# B&R Automation Studio project NAELD004C00R10L518F00 (part 33)

#### Act_Background.st
```iecst
(** 2020-05-26 **)
ACTION Act_Background:

	//Update Parameter
	IF bModuleOK = TRUE THEN

		tyParamInMove.diPosInUM		:= p_diMovePosInUM;
		tyParamInMove.diDistInUM	:= p_diMoveDistInUM;
		tyParamInMove.diVelInUMPS	:= p_diMoveVelInUMPS;
		tyParamInMove.diAcc			:= p_diMoveAcc;
		tyParamInMove.diDec			:= p_diMoveDec;

		fMotionCANUpdtDat(ADR(tyParamOut) , p_tyParamInConvert , tyParamOutDriver , tyParamInDriver , tyParamInMove , p_tyParamInHm , p_bDir, p_eNtParamMotorType);

		bWidthPosDiff	:= (tyParamOut.bIsHomed = FALSE) OR ((ABS((ABS(fAWWidthToPosInUM(p_diGoWidth , p_diWidthAtHmPos))) - tyParamOut.diActualPosInUM)) > 500);

		p_tyParamInConvert.diPitchInUM	:= fPitchCalc(p_diWidthOffsetInUM , p_diMaxWidthInUM , p_diMinWidthInUM , p_diPitchInUM);

		fbFullMovAbsBl.tyParamInConvert					:= p_tyParamInConvert;

		IF p_bDir = TRUE THEN
			bOpenSen	:= tyParamOut.bFwdLmtSen;
			bCloseSen	:= tyParamOut.bRevLmtSen;
		ELSE
			bOpenSen	:= tyParamOut.bRevLmtSen;
			bCloseSen	:= tyParamOut.bFwdLmtSen;
		END_IF

		CASE p_eNtParamMotorType OF
			DeltaAsdaA2:
				CASE tyParamOut.udiAxisErrID OF
					8976:	sAxisErrTxt	:= 'Over Current';
					12560:	sAxisErrTxt	:= 'Over Voltage';
					12576:	sAxisErrTxt	:= 'Under Voltage';
					12592:	sAxisErrTxt	:= 'Input Power Phase Loss';
					12816:	sAxisErrTxt	:= 'Regeneration Error';
					12848:	sAxisErrTxt	:= 'Overload';
					12849:	sAxisErrTxt	:= 'Pre-overload Warning';
					13056:	sAxisErrTxt	:= 'U,V,W Wiring Error';
					16912:	sAxisErrTxt	:= 'IGBT Temperature Error';
					21296:	sAxisErrTxt	:= 'Memory Error';
					21569:	sAxisErrTxt	:= 'Emergency Stop Activated';
					21570:	sAxisErrTxt	:= 'Forward Limit Switch Error';
					21571:	sAxisErrTxt	:= 'Reverse Limit Switch Error';
					21572:	sAxisErrTxt	:= 'Forward Software Limit';
					21573:	sAxisErrTxt	:= 'Reverse Software Limit';
					21760:	sAxisErrTxt	:= 'DSP Firmware Upgrade';
					25088:	sAxisErrTxt	:= 'CANopen SYNC Error';
					25360:	sAxisErrTxt	:= 'CANopen Data Initial Error';
					25376:	sAxisErrTxt	:= 'Adjustment Error';
					28961:	sAxisErrTxt	:= 'Motor Protection Error';
					28962:	sAxisErrTxt	:= 'Motor Error';
					29445:	sAxisErrTxt	:= 'Encoder Error';
					29446:	sAxisErrTxt	:= 'Encoder Output Error';
					29968:	sAxisErrTxt	:= 'Serial Communication Error';
					29984:	sAxisErrTxt	:= 'Serial Communication Time Out';
					33024:	sAxisErrTxt	:= 'CANbus Error (Bus-off)';
					33040:	sAxisErrTxt	:= 'CANopen SDO receive buffer overrun';
					33056:	sAxisErrTxt	:= 'CANbus Error (Warning)';
					33072:	sAxisErrTxt	:= 'Node Guarding or Heartbeat Error';
					33280:	sAxisErrTxt	:= 'CANopen PDO Object Error';
					33792:	sAxisErrTxt	:= 'Over Speed';
					34304:	sAxisErrTxt	:= 'Abnormal Pulse Control Command';
					34320:	sAxisErrTxt	:= 'Full Closed Loop Excessive Deviation';
					34321:	sAxisErrTxt	:= 'Excessive Deviation';
				END_CASE

			SchneiderLexium28:
				CASE tyParamOut.udiAxisErrID OF
					8724:	sAxisErrTxt	:= 'Over Current';
					8976:	sAxisErrTxt	:= 'Motor Overload';
					8977:	sAxisErrTxt	:= 'Drive overload (foldback)';
					9088:	sAxisErrTxt	:= 'Calculated offsets for current sensors out OF range';
					9089:	sAxisErrTxt := 'Motor phase missing';
					9090:	sAxisErrTxt := 'Overcurrent detected at one OF the digital outputs';
					12560:	sAxisErrTxt	:= 'DC Bus Over Voltage';
					12576:	sAxisErrTxt	:= 'DC Bus Under Voltage';
					12672:	sAxisErrTxt	:= 'Braking Resistor Overload';
					12673:	sAxisErrTxt	:= 'Safety function Safe Torque Off (STO) triggered';
					12674:	sAxisErrTxt	:= 'DC bus voltage measurement';
					12675:	sAxisErrTxt	:= 'Missing mains supply, undervoltage mains supply';
					12676:	sAxisErrTxt := 'The encoder supply voltage has dropped under operational value';
					12677:	sAxisErrTxt := 'The multi turn encoder battery voltage has dropped under 3 Vdc';
					12678:	sAxisErrTxt := 'Internal position synchronization error	detected between the multi turn AND the single turn modules';
					12679:	sAxisErrTxt := 'Generic error code of the multi turn module is detected';
					12697:	sAxisErrTxt := 'Braking resistor overload';
					16512:	sAxisErrTxt	:= 'Drive overtemperature (IPM)';
					16513:	sAxisErrTxt	:= 'Drive overtemperature (controller)';
					16534:	sAxisErrTxt := 'Temperature sensor inoperative';
					17168:	sAxisErrTxt	:= 'Power stage overtemperature';
					17280:	sAxisErrTxt := 'The encoder temperature is too high';
					17424:	sAxisErrTxt	:= 'Motor overtemperature';
					21808:	sAxisErrTxt	:= 'System error detected (nonvolatilememory)';
					21893:	sAxisErrTxt	:= 'Error detected in non-volatile memory';
					21889:	sAxisErrTxt	:= 'System error detected (nonvolatile memory)';
					21890:	sAxisErrTxt	:= 'System error detected (CAN power supply)';
					21891:	sAxisErrTxt	:= 'System error detected (selftest)';
					21894:	sAxisErrTxt	:= 'System error detected (NV ACCESS)';
					25472:	sAxisErrTxt	:= 'Target position rejected';
					25985:	sAxisErrTxt	:= 'System error detected(FPGA)';
					28816:	sAxisErrTxt	:= 'System error detected (FPGA does NOT match firmware)';
					28817:	sAxisErrTxt	:= 'Emergency Stop Activated';
					28961:	sAxisErrTxt := 'Motor blocked';
					29080:	sAxisErrTxt := 'Commutation error detected';
					29568:  sAxisErrTxt	:= 'Error detected in communication with motor encoder';
					29574:	sAxisErrTxt	:= 'Drive is not synchronous wit master cycle';
					29581:	sAxisErrTxt := 'System error detected (encoder)';
					29587:	sAxisErrTxt	:= 'Encoder overvoltage or overcurrent';
					29592:	sAxisErrTxt := 'The returned position value are no longer considered valid';
					29593:	sAxisErrTxt := 'The multi turn encoder requires an explicit configuration command';
					30081:	sAxisErrTxt := 'Target position rejected';
					30082:	sAxisErrTxt := 'No target values received via the fieldbus';
					33072:	sAxisErrTxt	:= 'CANopen: Heartbeat error detected';
					33296:	sAxisErrTxt := 'R_PDO is too short';
					33921:	sAxisErrTxt	:= 'Actual Motor Velocity Too High';
					33553:	sAxisErrTxt	:= 'Motor torque too high FOR an excessive period OF time';
					33664:	sAxisErrTxt := 'Unstable current loop';
					33922:	sAxisErrTxt := 'Velocity deviation too high';
					34321:	sAxisErrTxt	:= 'Position deviation too high';
					34432:	sAxisErrTxt := 'Position deviation via signal output function MC_OK';
					34441:	sAxisErrTxt := 'Position deviation too high (following error)';
					61568:	sAxisErrTxt	:= 'Fieldbus: Communication	error detected';
					65282:	sAxisErrTxt	:= 'Not possible to read data of electronic motor nameplate';
					65296:	sAxisErrTxt	:= 'Forward Limit Switch Error';
					65297:	sAxisErrTxt	:= 'Reverse Limit Switch Error';
					65281:	sAxisErrTxt := 'System error detected';
					65298:	sAxisErrTxt	:= 'Forward Software Limit';
					65299:	sAxisErrTxt	:= 'Reverse Software Limit';
					65301:	sAxisErrTxt := 'The encoder firmware cannot operate on the provided hardware';

				END_CASE

			EstunPronet:
				CASE tyParamOut.udiAxisErrID OF
					65281:	sAxisErrTxt	:= 'Parameter breakdown';//A01
					65282:	sAxisErrTxt	:= 'AD shift channels breakdown';
					65283:	sAxisErrTxt	:= 'Overspeed';
					65284:	sAxisErrTxt	:= 'Overload';
					65285:	sAxisErrTxt := 'Position error counteroverflow ';
					65286:	sAxisErrTxt := 'Position error pulse overflow';
					65287:	sAxisErrTxt	:= 'The setting of electronic gear or given pulse frequency is not reasonable';
					65288:	sAxisErrTxt	:= 'The 1st channel of current detection is wrong.';
					65289:	sAxisErrTxt	:= 'The 2nd channel of current detection is wrong.';
					65290:	sAxisErrTxt	:= 'Incremental Encoder is break off.';//A10
					65292:	sAxisErrTxt	:= 'Overcurrent';
					65293:	sAxisErrTxt	:= 'Overvoltage';
					65294:	sAxisErrTxt	:= 'Undervoltage';
					65295:	sAxisErrTxt := 'Bleeder resistor error';
					65296:	sAxisErrTxt := 'Regeneration error';
					65297:	sAxisErrTxt := 'Resolver error';
					65298:	sAxisErrTxt := 'IGBT superheat alarm';
					65299:	sAxisErrTxt := 'Motor overheat alarm';
					65300:	sAxisErrTxt := 'Power line phase shortage';//A20
					65301:	sAxisErrTxt	:= 'Instantaneous power off alarm';
					65302:	sAxisErrTxt	:= 'Motor temperature detection sensor is break off.';
					65303:	sAxisErrTxt := 'Brake overcurrent alarm';//A23
					65305:	sAxisErrTxt := 'Motor power line U overcurrent';//A25
					65306:	sAxisErrTxt := 'Motor power line V overcurrent';//A26
					65307:	sAxisErrTxt := 'Motor power line W overcurrent';//A27
					65322:	sAxisErrTxt	:= 'Servomotor type error';//A42
					65323:	sAxisErrTxt	:= 'Servo drive type error';
					65325:	sAxisErrTxt	:= 'Absolute encoder multiturn information error';
					65326:	sAxisErrTxt	:= 'Absolute encoder multiturn information overflow';
					65327:	sAxisErrTxt	:= 'Battery voltage below 2.5V';
					65328:	sAxisErrTxt	:= 'Battery voltage below 3.1V';//A48
					65330:	sAxisErrTxt := 'Serial encoder communication overtime ';//A50
					65331:	sAxisErrTxt := 'Absolute encoder overspeed alarm detected';
					65332:  sAxisErrTxt	:= 'Absolute state of serial encoder error';
					65333:	sAxisErrTxt	:= 'Serial encoder calcaution error';
					65334:	sAxisErrTxt := 'Parity bit or end bit in serial encoder control domain error';
					65335:	sAxisErrTxt	:= 'Serial encoder communication data checking error';
					65336:	sAxisErrTxt := 'End bit in serial encoder control domain error';
					65338:	sAxisErrTxt := 'Serial encoder data empty';
					65339:	sAxisErrTxt := 'Serial encoder data format error';
					65340:	sAxisErrTxt := 'Communication module not detected ';//A60
					65341:	sAxisErrTxt := 'Communication unsuccessful';
					65342:	sAxisErrTxt := 'Servo drive can not receive the period data of communication module ';
					65343:	sAxisErrTxt := 'Communication module can not receive the servo drive response data.';
					65344:	sAxisErrTxt := 'Communication module and bus connectionless';
					65346:	sAxisErrTxt := 'CAN communication abnormal';
					65347:	sAxisErrTxt := 'Receiving heartbeat timeout';
					65349:	sAxisErrTxt := 'Synchronization signal monitoring cycle is longer than setting';
					65362: sAxisErrTxt	:= 'Torque output alarm';
				END_CASE
		END_CASE

	ELSE

		tyParamOut.bAxisErr			:= FALSE;
		tyParamOut.bFwdLmtSen		:= FALSE;
		tyParamOut.bInPos			:= FALSE;
		tyParamOut.bIsHomed			:= FALSE;
		tyParamOut.bPosDiff			:= TRUE;
		tyParamOut.bPwrOn			:= FALSE;
		tyParamOut.bRevLmtSen		:= FALSE;
		tyParamOut.bStopped			:= TRUE;
		tyParamOut.diActualPosInUM	:= 0;
		tyParamOut.diHmAcc			:= 0;
		tyParamOut.diHmSpdForSwitch	:= 0;
		tyParamOut.diHmSpdForZero	:= 0;
		tyParamOut.diProfileAcc		:= 0;
		tyParamOut.diProfileDec		:= 0;
		tyParamOut.udiAxisErrID		:= 0;

		bWidthPosDiff				:= TRUE;

	END_IF

	//Abnormal Movement
	IF eStatus1 <> Error THEN
		IF p_bOps = TRUE AND eStatus = Idle THEN
			IF (ABS(tyParamOut.diActualPosInUM - diActualPosInUMOld) > 2000) AND (ABS(tyParamOut.diActualPosInUM - diActualPosInUMOld) < 10000) THEN
				eStatus1	:= Error;
				udiStatus1	:= 10000;	//Axis Move Abnormally By External Force

				fMotionCANRstCtrlWord(ADR(tyParamOutDriver));
				p_eAct	:= AWActIdle;
				eStat	:= AWActIdle;
			END_IF
		ELSE
			diActualPosInUMOld	:= tyParamOut.diActualPosInUM;
		END_IF
	END_IF

	//Reset Error
	IF (eStatus1 = Error) AND bRstErr THEN
		eStatus1	:= Idle;
		udiStatus1	:= 0;
	END_IF

	//Request Position To Movement Out Of Range
	IF p_bOps
		AND((tyParamInMove.diPosInUM < p_diMinAbsPosInUM) OR (tyParamInMove.diPosInUM > p_diMaxAbsPosInUM))
		AND (eStatus2 <> Error) THEN
		eStatus2	:= Error;
		udiStatus2	:= 10029;	//Request Absolute Position Out Of Range

		fMotionCANRstCtrlWord(ADR(tyParamOutDriver));
		p_eAct	:= AWActIdle;
		eStat	:= AWActIdle;
	END_IF

	//Reset Error
	IF (eStatus2 = Error) AND bRstErr THEN
		eStatus2	:= Idle;
		udiStatus2	:= 0;
	END_IF

	//Sensor Interrupt
	IF (bNotInterruptible = TRUE OR bJogging) AND eStatus3 <> Error THEN

		IF p_bInletSensor = TRUE THEN
			eStatus3	:= Error;
			udiStatus3	:= 10030;	//Inlet Sensor Interrupt Auto Width Movement

			fMotionCANRstCtrlWord(ADR(tyParamOutDriver));
			p_eAct	:= AWActIdle;
			eStat	:= AWActIdle;

		ELSIF p_bOutletSensor = TRUE THEN
			eStatus3	:= Error;
			udiStatus3	:= 10031;	//Outlet Sensor Interrupt Auto Width Movement

			fMotionCANRstCtrlWord(ADR(tyParamOutDriver));
			p_eAct	:= AWActIdle;
			eStat	:= AWActIdle;

		ELSIF p_bClearSensor = TRUE THEN
			eStatus3	:= Error;
			udiStatus3	:= 10032;	//Clear Sensor Interrupt Auto Width Movement

			fMotionCANRstCtrlWord(ADR(tyParamOutDriver));
			p_eAct	:= AWActIdle;
			eStat	:= AWActIdle;

		ELSIF p_bMiddleSensor = TRUE THEN
			eStatus3	:= Error;
			udiStatus3	:= 10033;	//Middle Sensor Interrupt Auto Width Movement

			fMotionCANRstCtrlWord(ADR(tyParamOutDriver));
			p_eAct	:= AWActIdle;
			eStat	:= AWActIdle;

		ELSIF p_bInterruptSensor = TRUE THEN
			eStatus3	:= Error;
			udiStatus3	:= 10034;	//Sensor Interrupt Auto Width Movement

			fMotionCANRstCtrlWord(ADR(tyParamOutDriver));
			p_eAct	:= AWActIdle;
			eStat	:= AWActIdle;

		ELSIF p_bCloseInterruptSensor = TRUE AND bJogOpen = FALSE THEN
			eStatus3	:= Error;
			udiStatus3	:= 10047;	//Sensor Interrupt Auto Width Movement

			fMotionCANRstCtrlWord(ADR(tyParamOutDriver));
			p_eAct	:= AWActIdle;
			eStat	:= AWActIdle;

		ELSIF p_bOpenInterruptSensor = TRUE AND bJogClose = FALSE THEN
			eStatus3	:= Error;
			udiStatus3	:= 10048;	//Sensor Interrupt Auto Width Movement

			fMotionCANRstCtrlWord(ADR(tyParamOutDriver));
			p_eAct	:= AWActIdle;
			eStat	:= AWActIdle;
		END_IF

	END_IF

	//Reset Error
	IF (eStatus3 = Error AND bRstErr)
		OR (p_bOpenInterruptSensor AND eStat = AWActJogClose)
		OR (p_bCloseInterruptSensor AND eStat = AWActJogOpen)
		THEN
		eStatus3	:= Idle;
		udiStatus3	:= 0;
	END_IF

	IF bRstErr THEN
		udiStatus	:= 0;
		bJogging	:= FALSE;
		bJogClose	:= FALSE;
		bJogOpen	:= FALSE;
	END_IF

	fbServoModuleOk(IN:= bModuleOK);
	fbServoModuleNotOk(IN:= bModuleOK = FALSE);
	IF fbServoModuleNotOk.Q AND udiStatus <> 10001 THEN

		bModuleNotOK		:= TRUE;
		bModuleNotOKLock	:= TRUE;
		usiRstStep	:= 0;
		tyParamOutDriver.uiCtrlword_6040	:= 0;
		tyParamOutDriver.siModOfOpt_6060	:= 0;
		tyParamOutDriver.diTargetPos_607A	:= 0;
		tyParamOutDriver.udiMoveSpd_6081	:= 0;
		tyParamOutDriver.siHmMethod_6098	:= 0;
		tyParamOutDriver.diJogVel_60FF		:= 0;

		CASE p_eNtParamMotorType OF

			DeltaAsdaA2:
				fbModuleOK(bModuleOK:= FALSE);
				IF eStatus = Idle THEN
					eAct	:= AWActRstNode;
				END_IF

				IF (eStatus = Done OR eStatus = Error)AND eStat = AWActRstNode THEN

					eAct	:= AWActIdle;
				END_IF

			EstunPronet:
				fbModuleOK(bModuleOK:= FALSE);
				IF eStatus = Idle THEN
					eAct	:= AWActRstNode;
				END_IF

				IF (eStatus = Done OR eStatus = Error)AND eStat = AWActRstNode THEN

					eAct	:= AWActIdle;
				END_IF

			SchneiderLexium28:
			// Do Nothing
		END_CASE

	ELSIF bModuleNotOK = TRUE AND fbServoModuleOk.Q THEN

		CASE usiRstStep OF

			0:
				IF eStatus = Idle THEN
					eAct	:= AWActRstAxisErr;
				END_IF

				IF eStatus = Done AND eStat = AWActRstAxisErr THEN
					eAct	:= AWActIdle;
					usiRstStep	:= 4;
				END_IF

			4: tyParamOutDriver.siModOfOpt_6060 := 1;
				usiRstStep	:= 5;

			5: tyParamOutDriver.siModOfOpt_6060 := 1;
				fbRstNodeTimer(IN:=TRUE);

				IF tyParamInDriver.siModOfOptDisp_6061 = 1 THEN
					usiRstStep	:= 6;
					fbRstNodeTimer(IN:=FALSE);
				ELSIF fbRstNodeTimer.Q THEN
					usiRstStep	:= 8;
					fbRstNodeTimer(IN:=FALSE);
				END_IF

			6: tyParamOutDriver.siModOfOpt_6060 := 6;
				fbRstNodeTimer(IN:=FALSE);
				usiRstStep	:= 7;

			7: tyParamOutDriver.siModOfOpt_6060 := 6;
				fbRstNodeTimer(IN:=TRUE);

				IF tyParamInDriver.siModOfOptDisp_6061 = 6 THEN
					usiRstStep	:= 10;
					fbRstNodeTimer(IN:=FALSE);
				ELSIF fbRstNodeTimer.Q THEN
					usiRstStep	:= 9;
					fbRstNodeTimer(IN:=FALSE);
				END_IF

			8:	fbModuleOK(bEn := TRUE, bModuleOK:= FALSE);
				fbRstNodeTimer(IN:=FALSE);
				usiRstStep	:= 9;

			9:	fbModuleOK(bModuleOK:= FALSE);
				IF eStatus = Idle THEN
					eAct	:=AWActRstNode;
				END_IF

				IF eStatus = Done AND eStat = AWActRstNode THEN
					usiRstStep	:= 0;
					eAct		:= AWActIdle;
				END_IF

			10:IF eStatus = Idle THEN
					eAct	:= AWActRstAxisErr;
				END_IF

				IF eStatus = Done AND eStat = AWActRstAxisErr THEN
					eAct			:=AWActIdle;
					usiRstStep	:= 11;
				END_IF

			11:

				IF eStatus = Idle THEN
					eAct	:= AWActSDOWrite;
				END_IF

				IF eStatus = Done AND eStat = AWActSDOWrite THEN
					eAct			:= AWActIdle;
					usiRstStep	:= 13;

				ELSIF udiStatus = 10028 THEN
					eAct			:= AWActIdle;
					usiRstStep	:= 0;
				END_IF

			13: bModuleNotOK	:= FALSE;
				usiRstStep	:= 0;
		END_CASE
	ELSE
		eAct	:= AWActIdle;

	END_IF

	IF tyParamOut.bPosDiff = FALSE THEN
		tyParamOutDriver.uiCtrlword_6040.4	:= FALSE;
	END_IF

END_ACTION
```

#### Act_InitGlobal.st
```iecst
(** 2019-04-09 **)
ACTION Act_InitGlobal:

	(* Always Change If Project Change *)

	//Pass Data To Link
	p_bLinkOpsRun ACCESS p_OpsRun;
	p_bLinkStartupRun ACCESS p_StartupRun;
	p_diLinkProdSelWidth ACCESS p_ProdRcpCurrRcp2Width;
	p_diLinkPshrOffset ACCESS p_ProdRcpCurrRcp2PshrOffset;
	p_diLinkMnlGoWidth ACCESS p_UIMnlAWPushOrPullerGoWidth;
	p_bLinkSafetyRelay ACCESS p_DISafetyRlySig;

	//Pass Data To Internal Use
	p_udiRstErr ACCESS p_RstErrReset;
	p_bManual ACCESS p_UIMnlMod;
	p_bEn ACCESS p_DISimServoEn;
	p_bPrep ACCESS p_NtParamAWPusherPrep;
	p_bDis ACCESS p_McParamAWPusherDis;
	p_bOps ACCESS p_OpsStatusRun;
	p_diWidthAtHmPos ACCESS p_McParamAWPusherAtHmPos;
	p_tyTuning ACCESS p_NtParamAWPushPulTuning;
	p_diJogVelInUMPS ACCESS p_UIMnlAWPushOrPullerJogSpd;
	p_diMovePosInUM ACCESS p_UIMnlAWPushOrPullerTargetPos;
	p_diMoveDistInUM ACCESS p_UIMnlAWPushOrPullerStepSize;
	p_bUITeachServo ACCESS p_UITeachServo;
	p_diMoveAcc ACCESS p_NtParamAWPushPulAcc;
	p_diMoveDec ACCESS p_NtParamAWPushPulDec;
	p_diMinWidthInUM ACCESS p_NtParamProdRcpMinWidth;
	p_diMaxWidthInUM ACCESS p_NtParamProdRcpMaxWidth;
	p_diWidthOffsetInUM ACCESS p_NtParamPushPulAWidthOffset;
	p_bInletSensor ACCESS p_DIConvLftSen;
	p_bOutletSensor ACCESS p_DIConvRgtSen;
	p_bDir ACCESS p_NtParamAWPushPulDir;
	p_bDirBl ACCESS p_NtParamAWPushPulDirBl;
	p_usiNode ACCESS p_NtParamAWPushPulNode;
	p_sDevice ACCESS p_NtParamAWPushPulDevice;
	p_sProgNm ACCESS p_NtParamAWPushPulProgNm;
	p_diMoveBacklashDistInUM ACCESS p_NtParamAWPushPulMovBlDistInUM;
	p_diPitchInUM ACCESS p_NtParamAWPushPulPitchInUM;
	p_tyParamInHm ACCESS p_NtParamAWPushPulParamInHm;
	p_tyParamInConvert ACCESS p_NtParamAWPushPulParamInConvert;
	p_bNtSettingsLoadDone ACCESS p_StartupNtSettingsLoadDone;
	p_eNtParamMotorType ACCESS p_NtParamAWPushPulMotorType;

	p_bInletShutterCloseRS ACCESS p_DIInShutterCloseRS;
	p_bOutletShutterCloseRS ACCESS p_DIOutShutterCloseRS;
	p_bProjInletShutPrep ACCESS p_NtParamProjInletShutPrep;
	p_bProjOutletShutPrep ACCESS p_NtParamProjOutletShutPrep;
	p_bOutShutterDis ACCESS p_McParamOutShutterDis;
	p_bPullerRetSen ACCESS p_DIPullerRetRS;
	p_bPullerExtSen ACCESS p_DIPullerExtRS;
	(* Always Change If Project Change *)

END_ACTION
```

#### Act_Link.st
```iecst
(** 2019-03-29 **)
ACTION Act_Link:

	IF p_bManual = TRUE THEN
		p_diMoveVelInUMPS ACCESS p_UIMnlAWPushOrPullerNomSpd;
		IF p_diLinkMnlGoWidth < p_diWidthAtHmPos THEN
			p_diGoWidth := p_diWidthAtHmPos;
		ELSE
			p_diGoWidth	:= p_diLinkMnlGoWidth;
		END_IF

	ELSE

		p_diMoveVelInUMPS ACCESS p_NtParamAWPushPulAutoSpd;
		IF ((p_diLinkProdSelWidth/2) + p_diLinkPshrOffset) < p_diWidthAtHmPos THEN
			p_diGoWidth := p_diWidthAtHmPos+3000;
		ELSE
			//	p_diGoWidth := ((p_diLinkProdSelWidth/2) + p_diLinkPshrOffset)/2;
			IF p_diLinkPshrOffset = 0 THEN
				p_diGoWidth := (p_diLinkProdSelWidth/2) - 50000;
			ELSE
				p_diGoWidth := (p_diLinkProdSelWidth/2) + p_diLinkPshrOffset;
			END_IF
		END_IF

	END_IF

	IF p_bProjInletShutPrep = TRUE THEN
		IF p_bInletShutterCloseRS = FALSE OR p_bPullerRetSen = FALSE
			THEN
			bInterruptSensor1 := TRUE;
		ELSE
			bInterruptSensor1 := FALSE;
		END_IF
	ELSE
		bInterruptSensor1 := FALSE;
	END_IF

	IF p_bProjOutletShutPrep = TRUE AND p_bOutShutterDis = FALSE THEN
		IF p_bOutletShutterCloseRS = FALSE OR p_bPullerRetSen = FALSE
			THEN
			bInterruptSensor2 := TRUE;
		ELSE
			bInterruptSensor2 := FALSE;
		END_IF
	ELSE
		bInterruptSensor2 := FALSE;
	END_IF

	p_bInterruptSensor := bInterruptSensor2 OR bInterruptSensor1;// OR p_bLinkSafetyRelay = FALSE;

END_ACTION
```

#### Act_LinkAction.st
```iecst
(** 2019-10-21 **)
ACTION Act_LinkAction:

	IF eStatus = Idle THEN
		IF bModuleNotOK THEN
			p_eAct ACCESS ADR(eAct);
		ELSE
			IF p_bLinkStartupRun = TRUE THEN
				p_eAct ACCESS p_StartupAWPushPulAct;
			ELSIF p_bLinkOpsRun = TRUE THEN
				p_eAct ACCESS p_OpsTravLifLDAWPushPullAct;
			ELSIF p_bManual = TRUE THEN
				p_eAct ACCESS p_UIAWPushOrPullerAct;
			ELSE
				p_eAct ACCESS ADR(eAct);
			END_IF
		END_IF
	END_IF

	IF EDGENEG(p_bManual) OR EDGENEG(p_bLinkOpsRun) OR EDGENEG(p_bLinkStartupRun) THEN
		tyParamOutDriver.uiCtrlword_6040	:= 0;
	END_IF

END_ACTION
```

### Program Logical/CANOpenServo/Trav/Trav

#### InputRef.var
```iecst
(*2020-03-16*)
(**)
(*General*)
VAR
	p_eAct : REFERENCE TO eTravAction;
	p_udiRstErr : REFERENCE TO UDINT;
	p_bPrep : REFERENCE TO BOOL;
	p_bEn : REFERENCE TO BOOL;
	p_bDis : REFERENCE TO BOOL;
END_VAR
(**)
(*Configuration*)
VAR
	p_bOps : REFERENCE TO BOOL;
	p_bManual : REFERENCE TO BOOL;
	p_diAPos : REFERENCE TO DINT;
	p_diBPos : REFERENCE TO DINT;
	p_diCPos : REFERENCE TO DINT;
	p_diDPos : REFERENCE TO DINT;
	p_diEPos : REFERENCE TO DINT;
	p_diFPos : REFERENCE TO DINT;
	p_diGPos : REFERENCE TO DINT;
	p_diHPos : REFERENCE TO DINT;
	p_tyTuning : REFERENCE TO tyMotionCANTuning;
	p_diJogVelInUMPS : REFERENCE TO DINT;
	p_diMovePosInUM : REFERENCE TO DINT;
	p_diMoveDistInUM : REFERENCE TO DINT;
	p_diMoveVelInUMPS : REFERENCE TO DINT;
	p_diMoveAcc : REFERENCE TO DINT;
	p_diMoveDec : REFERENCE TO DINT;
	p_diMinAbsPosInUM : REFERENCE TO DINT;
	p_diMaxAbsPosInUM : REFERENCE TO DINT;
	p_bInterruptSensor1 : REFERENCE TO BOOL;
	p_bInterruptSensor2 : REFERENCE TO BOOL;
	p_bInterruptSensor3 : REFERENCE TO BOOL;
	p_bInterruptSensor4 : REFERENCE TO BOOL;
	p_bInterruptSensor5 : REFERENCE TO BOOL;
	p_usiNode : REFERENCE TO USINT;
	p_bDir : REFERENCE TO BOOL;
	p_bNoIndexPulse : REFERENCE TO BOOL;
	p_sDevice : REFERENCE TO STRING[3];
	p_sProgNm : REFERENCE TO STRING[15];
	p_tyParamInHm : REFERENCE TO tyMotionCANParamInHm;
	p_tyParamInConvert : REFERENCE TO tyMotionCANParamInConvert;
	p_bNtSettingsLoadDone : REFERENCE TO BOOL;
	p_eNtParamMotorType : REFERENCE TO eServoMotorType;
	p_bProjInletShutPrep : REFERENCE TO BOOL;
	p_bProjOutletShutPrep : REFERENCE TO BOOL;
	p_bOutletShutterCloseRS : REFERENCE TO BOOL;
	p_bOutShutterDis : REFERENCE TO BOOL;
	p_bInletShutterCloseRS : REFERENCE TO BOOL;
	p_bPullerExtSen : REFERENCE TO BOOL;
	p_bPullerRetSen : REFERENCE TO BOOL;
	p_bPullerRotHmRS : REFERENCE TO BOOL;
	p_bDIConvClrSen : REFERENCE TO BOOL;
	p_bDIConvLftSen : REFERENCE TO BOOL;
END_VAR
```

#### InputRef_Link.var
```iecst
(*2019-04-09*)
(**)
(*External Data*)
VAR
	p_bLinkOpsRun : REFERENCE TO BOOL;
	p_bLinkStartupRun : REFERENCE TO BOOL;
	p_bSimu : REFERENCE TO BOOL;
	p_diLinkAPos : REFERENCE TO DINT;
	p_diLinkBPos : REFERENCE TO DINT;
	p_diLinkCPos : REFERENCE TO DINT;
	p_diLinkGPos : REFERENCE TO DINT;
	p_diLinkAPos1 : REFERENCE TO DINT;
	p_diLinkBPos1 : REFERENCE TO DINT;
	p_diLinkCPos1 : REFERENCE TO DINT;
	p_diLinkGPos1 : REFERENCE TO DINT;
	p_bLinkNtParamProjRotCylPrep : REFERENCE TO BOOL;
END_VAR
(**)
VAR
	p_eLinkMag : REFERENCE TO eLDMag;
	p_usiLinkMod : REFERENCE TO USINT;
	p_bLinkOpsTravLifULInDSPos : REFERENCE TO BOOL;
	p_bLinkOpsTravLifUSMagWidthChk : REFERENCE TO BOOL;
	p_bLinkNtParamProjDsFixToFixRail : REFERENCE TO BOOL;
	p_diLinkFixtoFixPosIn : REFERENCE TO DINT;
	p_diLinkMcParamTravPosB : REFERENCE TO DINT;
	p_tyProdRcpCurrRcp : REFERENCE TO tyProdRcpParam;
	p_bLinkSafetyRelay : REFERENCE TO BOOL;
	p_bLinkProjLifterMagPlatform : REFERENCE TO BOOL;
	p_bLinkTravGotoChkPt : REFERENCE TO BOOL;
	p_diLinkTravGotoChkPtDist1 : REFERENCE TO DINT;
	p_diLinkTravGotoChkPtDist2 : REFERENCE TO DINT;
	p_diLinkTravGotoChkPtDist3 : REFERENCE TO DINT;
	p_diLaneBOffset : REFERENCE TO DINT;
END_VAR
```

#### Local.var
```iecst
(*2020-03-16*)
(**)
(*Local Action, State & Status*)
VAR
	eAct : eTravAction := TravActIdle;
	eStat : eTravAction := TravActIdle;
	eMainStatus : eFBStatus := Idle;
	eStatus : eFBStatus := Idle;
	eStatus1 : eFBStatus := Idle;
	eStatus2 : eFBStatus := Idle;
	eStatus3 : eFBStatus := Idle;
	udiStatus : UDINT := 0;
	udiStatus1 : UDINT := 0;
	udiStatus2 : UDINT := 0;
	udiStatus3 : UDINT := 0;
	sStatTxt : STRING[200] := '';
	a_sStatText : ARRAY[0..50] OF STRING[200] := ['Idling','Going A Position','Going B Position','Going C Position','Going D Position','Going E Position','Going F Position','Going G Position','Going H Position','Full Homing','Powering On','Powering Off','Homing','Moving Absolute','Moving Relative','Jogging Front','Jogging Rear','Jogging Stop','Resetting Axis Error','Stopping','Writing SDO','Background Start Module OK Check','Background Stop Module OK Check',28('')];
END_VAR
(**)
(*Local Alarm*)
VAR
	tyAlmData : tyAlmDat;
	tyAlmData1 : tyAlmDat;
	tyAlmData2 : tyAlmDat;
	tyAlmData3 : tyAlmDat;
	a_tyAlmText : ARRAY[10000..10299] OF tyAlmTxt := [(sAlmText:='Axis Move Abnormally By External Force',sRcyText:='Servo Motor Abnormal Operation. Reset And Resume Operation. If The Problem Persists, Please Contact Nutek For A Possible Solution.'),(sAlmText:='CANOpen Communication Error, ModuleOK Not TRUE',sRcyText:='Fail While Read/Write Data. Reset The Error And Resume Operation.'),(sAlmText:='Power On Time Out While Going A Position',sRcyText:='Timeout Expired Before Operation Completed. Reset And Resume Operation.'),(sAlmText:='Homing Time Out While Going A Position',sRcyText:='Timeout Expired Before Operation Completed. Reset And Resume Operation.'),(sAlmText:='Move Absolute Time Out While Going A Position',sRcyText:='Timeout Expired Before Operation Completed. Reset And Resume Operation.'),(sAlmText:='Stop Motion Time Out While Going A Position',sRcyText:='Timeout Expired Before Operation Completed. Reset And Resume Operation.'),(sAlmText:='Axis Error Reset Failed While Going A Position',sRcyText:='Axis Error Reset Failed. Please Retry Again Reset Operation. If The Problem Persists, Please Contact Nutek For A Possible Solution.'),(sAlmText:='Axis Error Occur In Move Absolute While Going A Position',sRcyText:='Servo Motor Abnormal Operation. Reset And Resume Operation. If The Problem Persists, Please Contact Nutek For A Possible Solution.'),(sAlmText:='Axis Error Occur In Homing While Going A Position',sRcyText:='Servo Motor Abnormal Operation. Reset And Resume Operation. If The Problem Persists, Please Contact Nutek For A Possible Solution.'),(sAlmText:='Homing Done But Home Flag Is Not Activated While Going A Position',sRcyText:='Servo Motor Abnormal Operation. Reset And Resume Operation. If The Problem Persists, Please Contact Nutek For A Possible Solution.'),(sAlmText:='Forward Limit Activated In Homing While Going A Position',sRcyText:='Forward Limit Switch Is Activated. Reset The Error By Operate The Motor Backwards.'),(sAlmText:='Reverse Limit Activated In Homing While Going A Position',sRcyText:='Reverse Limit Switch Is Activated. Reset The Error By Operate The Motor Backwards.'),(sAlmText:='Forward Limit Activated In Move Absolute While Going A Position',sRcyText:='Forward Limit Switch Is Activated. Reset The Error By Operate The Motor Backwards.'),(sAlmText:='Reverse Limit Activated In Move Absolute While Going A Position',sRcyText:='Reverse Limit Switch Is Activated. Reset The Error By Operate The Motor Backwards.'),(sAlmText:='Power On Time Out While Full Homing',sRcyText:='Timeout Expired Before Operation Completed. Reset And Resume Operation.'),(sAlmText:='Homing Time Out While Full Homing',sRcyText:='Timeout Expired Before Operation Completed. Reset And Resume Operation.'),(sAlmText:='Stop Motion Time Out While Full Homing',sRcyText:='Timeout Expired Before Operation Completed. Reset And Resume Operation.'),(sAlmText:='Axis Error Reset Failed While Full Homing',sRcyText:='Axis Error Reset Failed. Please Retry Again Reset Operation. If The Problem Persists, Please Contact Nutek For A Possible Solution.'),(sAlmText:='Axis Error Occur In Homing While Full Homing',sRcyText:='Servo Motor Abnormal Operation. Reset And Resume Operation. If The Problem Persists, Please Contact Nutek For A Possible Solution.'),(sAlmText:='Homing Done But Home Flag Is Not Activated While Full Homing',sRcyText:='Servo Motor Abnormal Operation. Reset And Resume Operation. If The Problem Persists, Please Contact Nutek For A Possible Solution.'),(sAlmText:='Forward Limit Activated In Homing While Full Homing',sRcyText:='Forward Limit Switch Is Activated. Reset The Error By Operate The Motor Backwards.'),(sAlmText:='Reverse Limit Activated In Homing While Full Homing',sRcyText:='Reverse Limit Switch Is Activated. Reset The Error By Operate The Motor Backwards.'),(sAlmText:='Power On Time Out',sRcyText:='Timeout Expired Before Operation Completed. Reset And Resume Operation.'),(sAlmText:='Power Off Time Out',sRcyText:='Timeout Expired Before Operation Completed. Reset And Resume Operation.'),(sAlmText:='Homing Time Out',sRcyText:='Timeout Expired Before Operation Completed. Reset And Resume Operation.'),(sAlmText:='Move Absolute Time Out',sRcyText:='Timeout Expired Before Operation Completed. Reset And Resume Operation.'),(sAlmText:='Move Relative Time Out',sRcyText:='Timeout Expired Before Operation Completed. Reset And Resume Operation.'),(sAlmText:='Stop Motion Time Out',sRcyText:='Timeout Expired Before Operation Completed. Reset And Resume Operation.'),(sAlmText:='SDO Write Error',sRcyText:='Fail While Write Data. Reset The Error And Resume Operation.'),(sAlmText:='Power On Time Out While Going B Position',sRcyText:='Timeout Expired Before Operation Completed. Reset And Resume Operation.'),(sAlmText:='Homing Time Out While Going B Position',sRcyText:='Timeout Expired Before Operation Completed. Reset And Resume Operation.'),(sAlmText:='Move Absolute Time Out While Going B Position',sRcyText:='Timeout Expired Before Operation Completed. Reset And Resume Operation.'),(sAlmText:='Stop Motion Time Out While Going B Position',sRcyText:='Timeout Expired Before Operation Completed. Reset And Resume Operation.'),(sAlmText:='Axis Error Reset Failed While Going B Position',sRcyText:='Axis Error Reset Failed. Please Retry Again Reset Operation. If The Problem Persists, Please Contact Nutek For A Possible Solution.'),(sAlmText:='Axis Error Occur In Move Absolute While Going B Position',sRcyText:='Servo Motor Abnormal Operation. Reset And Resume Operation. If The Problem Persists, Please Contact Nutek For A Possible Solution.'),(sAlmText:='Axis Error Occur In Homing While Going B Position',sRcyText:='Servo Motor Abnormal Operation. Reset And Resume Operation. If The Problem Persists, Please Contact Nutek For A Possible Solution.'),(sAlmText:='Homing Done But Home Flag Is Not Activated While Going B Position',sRcyText:='Servo Motor Abnormal Operation. Reset And Resume Operation. If The Problem Persists, Please Contact Nutek For A Possible Solution.'),(sAlmText:='Forward Limit Activated In Homing While Going B Position',sRcyText:='Forward Limit Switch Is Activated. Reset The Error By Operate The Motor Backwards.'),(sAlmText:='Reverse Limit Activated In Homing While Going B Position',sRcyText:='Reverse Limit Switch Is Activated. Reset The Error By Operate The Motor Backwards.'),(sAlmText:='Forward Limit Activated In Move Absolute While Going B Position',sRcyText:='Forward Limit Switch Is Activated. Reset The Error By Operate The Motor Backwards.'),(sAlmText:='Reverse Limit Activated In Move Absolute While Going B Position',sRcyText:='Reverse Limit Switch Is Activated. Reset The Error By Operate The Motor Backwards.'),(sAlmText:='Sensor Interrupt Movement',sRcyText:='Clear Interrupt Sensor And Resume Operation.'),35((0)),(sAlmText:='Request Absolute Position Out Of Range',sRcyText:='Request Absolute Position Does Not Fall Within The Expected Range.'),(sAlmText:='Power On Time Out While Going C Position',sRcyText:='Timeout Expired Before Operation Completed. Reset And Resume Operation.'),(sAlmText:='Homing Time Out While Going C Position',sRcyText:='Timeout Expired Before Operation Completed. Reset And Resume Operation.'),(sAlmText:='Move Absolute Time Out While Going C Position',sRcyText:='Timeout Expired Before Operation Completed. Reset And Resume Operation.'),(sAlmText:='Stop Motion Time Out While Going C Position',sRcyText:='Timeout Expired Before Operation Completed. Reset And Resume Operation.'),(sAlmText:='Axis Error Reset Failed While Going C Position',sRcyText:='Axis Error Reset Failed. Please Retry Again Reset Operation. If The Problem Persists, Please Contact Nutek For A Possible Solution.'),(sAlmText:='Axis Error Occur In Move Absolute While Going C Position',sRcyText:='Servo Motor Abnormal Operation. Reset And Resume Operation. If The Problem Persists, Please Contact Nutek For A Possible Solution.'),(sAlmText:='Axis Error Occur In Homing While Going C Position',sRcyText:='Servo Motor Abnormal Operation. Reset And Resume Operation. If The Problem Persists, Please Contact Nutek For A Possible Solution.'),(sAlmText:='Homing Done But Home Flag Is Not Activated While Going C Position',sRcyText:='Servo Motor Abnormal Operation. Reset And Resume Operation. If The Problem Persists, Please Contact Nutek For A Possible Solution.'),(sAlmText:='Forward Limit Activated In Homing While Going C Position',sRcyText:='Forward Limit Switch Is Activated. Reset The Error By Operate The Motor Backwards.'),(sAlmText:='Reverse Limit Activated In Homing While Going C Position',sRcyText:='Reverse Limit Switch Is Activated. Reset The Error By Operate The Motor Backwards.'),(sAlmText:='Forward Limit Activated In Move Absolute While Going C Position',sRcyText:='Forward Limit Switch Is Activated. Reset The Error By Operate The Motor Backwards.'),(sAlmText:='Reverse Limit Activated In Move Absolute While Going C Position',sRcyText:='Reverse Limit Switch Is Activated. Reset The Error By Operate The Motor Backwards.'),(sAlmText:='Power On Time Out While Going D Position',sRcyText:='Timeout Expired Before Operation Completed. Reset And Resume Operation.'),(sAlmText:='Homing Time Out While Going D Position',sRcyText:='Timeout Expired Before Operation Completed. Reset And Resume Operation.'),(sAlmText:='Move Absolute Time Out While Going D Position',sRcyText:='Timeout Expired Before Operation Completed. Reset And Resume Operation.'),(sAlmText:='Stop Motion Time Out While Going D Position',sRcyText:='Timeout Expired Before Operation Completed. Reset And Resume Operation.'),(sAlmText:='Axis Error Reset Failed While Going D Position',sRcyText:='Axis Error Reset Failed. Please Retry Again Reset Operation. If The Problem Persists, Please Contact Nutek For A Possible Solution.'),(sAlmText:='Axis Error Occur In Move Absolute While Going D Position',sRcyText:='Servo Motor Abnormal Operation. Reset And Resume Operation. If The Problem Persists, Please Contact Nutek For A Possible Solution.'),(sAlmText:='Axis Error Occur In Homing While Going D Position',sRcyText:='Servo Motor Abnormal Operation. Reset And Resume Operation. If The Problem Persists, Please Contact Nutek For A Possible Solution.'),(sAlmText:='Homing Done But Home Flag Is Not Activated While Going D Position',sRcyText:='Servo Motor Abnormal Operation. Reset And Resume Operation. If The Problem Persists, Please Contact Nutek For A Possible Solution.'),(sAlmText:='Forward Limit Activated In Homing While Going D Position',sRcyText:='Forward Limit Switch Is Activated. Reset The Error By Operate The Motor Backwards.'),(sAlmText:='Reverse Limit Activated In Homing While Going D Position',sRcyText:='Reverse Limit Switch Is Activated. Reset The Error By Operate The Motor Backwards.'),(sAlmText:='Forward Limit Activated In Move Absolute While Going D Position',sRcyText:='Forward Limit Switch Is Activated. Reset The Error By Operate The Motor Backwards.'),(sAlmText:='Reverse Limit Activated In Move Absolute While Going D Position',sRcyText:='Reverse Limit Switch Is Activated. Reset The Error By Operate The Motor Backwards.'),(sAlmText:='Power On Time Out While Going E Position',sRcyText:='Timeout Expired Before Operation Completed. Reset And Resume Operation.'),(sAlmText:='Homing Time Out While Going E Position',sRcyText:='Timeout Expired Before Operation Completed. Reset And Resume Operation.'),(sAlmText:='Move Absolute Time Out While Going E Position',sRcyText:='Timeout Expired Before Operation Completed. Reset And Resume Operation.'),(sAlmText:='Stop Motion Time Out While Going E Position',sRcyText:='Timeout Expired Before Operation Completed. Reset And Resume Operation.'),(sAlmText:='Axis Error Reset Failed While Going E Position',sRcyText:='Axis Error Reset Failed. Please Retry Again Reset Operation. If The Problem Persists, Please Contact Nutek For A Possible Solution.'),(sAlmText:='Axis Error Occur In Move Absolute While Going E Position',sRcyText:='Servo Motor Abnormal Operation. Reset And Resume Operation. If The Problem Persists, Please Contact Nutek For A Possible Solution.'),(sAlmText:='Axis Error Occur In Homing While Going E Position',sRcyText:='Servo Motor Abnormal Operation. Reset And Resume Operation. If The Problem Persists, Please Contact Nutek For A Possible Solution.'),(sAlmText:='Homing Done But Home Flag Is Not Activated While Going E Position',sRcyText:='Servo Motor Abnormal Operation. Reset And Resume Operation. If The Problem Persists, Please Contact Nutek For A Possible Solution.'),(sAlmText:='Forward Limit Activated In Homing While Going E Position',sRcyText:='Forward Limit Switch Is Activated. Reset The Error By Operate The Motor Backwards.'),(sAlmText:='Reverse Limit Activated In Homing While Going E Position',sRcyText:='Reverse Limit Switch Is Activated. Reset The Error By Operate The Motor Backwards.'),(sAlmText:='Forward Limit Activated In Move Absolute While Going E Position',sRcyText:='Forward Limit Switch Is Activated. Reset The Error By Operate The Motor Backwards.'),(sAlmText:='Reverse Limit Activated In Move Absolute While Going E Position',sRcyText:='Reverse Limit Switch Is Activated. Reset The Error By Operate The Motor Backwards.'),(sAlmText:='Power On Time Out While Going F Position',sRcyText:='Timeout Expired Before Operation Completed. Reset And Resume Operation.'),(sAlmText:='Homing Time Out While Going F Position',sRcyText:='Timeout Expired Before Operation Completed. Reset And Resume Operation.'),(sAlmText:='Move Absolute Time Out While Going F Position',sRcyText:='Timeout Expired Before Operation Completed. Reset And Resume Operation.'),(sAlmText:='Stop Motion Time Out While Going F Position',sRcyText:='Timeout Expired Before Operation Completed. Reset And Resume Operation.'),(sAlmText:='Axis Error Reset Failed While Going F Position',sRcyText:='Axis Error Reset Failed. Please Retry Again Reset Operation. If The Problem Persists, Please Contact Nutek For A Possible Solution.'),(sAlmText:='Axis Error Occur In Move Absolute While Going F Position',sRcyText:='Servo Motor Abnormal Operation. Reset And Resume Operation. If The Problem Persists, Please Contact Nutek For A Possible Solution.'),(sAlmText:='Axis Error Occur In Homing While Going F Position',sRcyText:='Servo Motor Abnormal Operation. Reset And Resume Operation. If The Problem Persists, Please Contact Nutek For A Possible Solution.'),(sAlmText:='Homing Done But Home Flag Is Not Activated While Going F Position',sRcyText:='Servo Motor Abnormal Operation. Reset And Resume Operation. If The Problem Persists, Please Contact Nutek For A Possible Solution.'),(sAlmText:='Forward Limit Activated In Homing While Going F Position',sRcyText:='Forward Limit Switch Is Activated. Reset The Error By Operate The Motor Backwards.'),(sAlmText:='Reverse Limit Activated In Homing While Going F Position',sRcyText:='Reverse Limit Switch Is Activated. Reset The Error By Operate The Motor Backwards.'),(sAlmText:='Forward Limit Activated In Move Absolute While Going F Position',sRcyText:='Forward Limit Switch Is Activated. Reset The Error By Operate The Motor Backwards.'),(sAlmText:='Reverse Limit Activated In Move Absolute While Going F Position',sRcyText:='Reverse Limit Switch Is Activated. Reset The Error By Operate The Motor Backwards.'),(sAlmText:='Power On Time Out While Going G Position',sRcyText:='Timeout Expired Before Operation Completed. Reset And Resume Operation.'),(sAlmText:='Homing Time Out While Going G Position',sRcyText:='Timeout Expired Before Operation Completed. Reset And Resume Operation.'),(sAlmText:='Move Absolute Time Out While Going G Position',sRcyText:='Timeout Expired Before Operation Completed. Reset And Resume Operation.'),(sAlmText:='Stop Motion Time Out While Going G Position',sRcyText:='Timeout Expired Before Operation Completed. Reset And Resume Operation.'),(sAlmText:='Axis Error Reset Failed While Going G Position',sRcyText:='Axis Error Reset Failed. Please Retry Again Reset Operation. If The Problem Persists, Please Contact Nutek For A Possible Solution.'),(sAlmText:='Axis Error Occur In Move Absolute While Going G Position',sRcyText:='Servo Motor Abnormal Operation. Reset And Resume Operation. If The Problem Persists, Please Contact Nutek For A Possible Solution.'),(sAlmText:='Axis Error Occur In Homing While Going G Position',sRcyText:='Servo Motor Abnormal Operation. Reset And Resume Operation. If The Problem Persists, Please Contact Nutek For A Possible Solution.'),(sAlmText:='Homing Done But Home Flag Is Not Activated While Going G Position',sRcyText:='Servo Motor Abnormal Operation. Reset And Resume Operation. If The Problem Persists, Please Contact Nutek For A Possible Solution.'),(sAlmText:='Forward Limit Activated In Homing While Going G Position',sRcyText:='Forward Limit Switch Is Activated. Reset The Error By Operate The Motor Backwards.'),(sAlmText:='Reverse Limit Activated In Homing While Going G Position',sRcyText:='Reverse Limit Switch Is Activated. Reset The Error By Operate The Motor Backwards.'),(sAlmText:='Forward Limit Activated In Move Absolute While Going G Position',sRcyText:='Forward Limit Switch Is Activated. Reset The Error By Operate The Motor Backwards.'),(sAlmText:='Reverse Limit Activated In Move Absolute While Going G Position',sRcyText:='Reverse Limit Switch Is Activated. Reset The Error By Operate The Motor Backwards.'),(sAlmText:='Power On Time Out While Going H Position',sRcyText:='Timeout Expired Before Operation Completed. Reset And Resume Operation.'),(sAlmText:='Homing Time Out While Going H Position',sRcyText:='Timeout Expired Before Operation Completed. Reset And Resume Operation.'),(sAlmText:='Move Absolute Time Out While Going H Position',sRcyText:='Timeout Expired Before Operation Completed. Reset And Resume Operation.'),(sAlmText:='Stop Motion Time Out While Going H Position',sRcyText:='Timeout Expired Before Operation Completed. Reset And Resume Operation.'),(sAlmText:='Axis Error Reset Failed While Going H Position',sRcyText:='Axis Error Reset Failed. Please Retry Again Reset Operation. If The Problem Persists, Please Contact Nutek For A Possible Solution.'),(sAlmText:='Axis Error Occur In Move Absolute While Going H Position',sRcyText:='Servo Motor Abnormal Operation. Reset And Resume Operation. If The Problem Persists, Please Contact Nutek For A Possible Solution.'),(sAlmText:='Axis Error Occur In Homing While Going H Position',sRcyText:='Servo Motor Abnormal Operation. Reset And Resume Operation. If The Problem Persists, Please Contact Nutek For A Possible Solution.'),(sAlmText:='Homing Done But Home Flag Is Not Activated While Going H Position',sRcyText:='Servo Motor Abnormal Operation. Reset And Resume Operation. If The Problem Persists, Please Contact Nutek For A Possible Solution.'),(sAlmText:='Forward Limit Activated In Homing While Going H Position',sRcyText:='Forward Limit Switch Is Activated. Reset The Error By Operate The Motor Backwards.'),(sAlmText:='Reverse Limit Activated In Homing While Going H Position',sRcyText:='Reverse Limit Switch Is Activated. Reset The Error By Operate The Motor Backwards.'),(sAlmText:='Forward Limit Activated In Move Absolute While Going H Position',sRcyText:='Forward Limit Switch Is Activated. Reset The Error By Operate The Motor Backwards.'),(sAlmText:='Reverse Limit Activated In Move Absolute While Going H Position',sRcyText:='Reverse Limit Switch Is Activated. Reset The Error By Operate The Motor Backwards.'),(sAlmText:='Request Absolute Position Out Of Range',sRcyText:='Request Absolute Position Does Not Fall Within The Expected Range.'),(sAlmText:='Sensor Interrupt Traverser Movement',sRcyText:='Operation Stop Due To The Interruption Of Sensor While Traverser Moving. Solve The Interruption To Resume Operation.'),148((0))];
END_VAR
(**)
(*Local Output*)
VAR
	tyParamOut : tyMotionCANParamOut;
	sAxisErrTxt : STRING[80];
	bAPosDiff : BOOL;
	bBPosDiff : BOOL;
	bCPosDiff : BOOL;
	bDPosDiff : BOOL;
	bEPosDiff : BOOL;
	bFPosDiff : BOOL;
	bGPosDiff : BOOL;
	bHPosDiff : BOOL;
	bJogging : BOOL;
	bFrontSen : BOOL;
	bRearSen : BOOL;
END_VAR
(**)
(*Local Input*)
VAR
	udiRstErr : UDINT := 0;
	bPrep : BOOL := TRUE;
	bEn : BOOL := TRUE;
	bDis : BOOL := FALSE;
	bOps : BOOL := FALSE;
	bManual : BOOL := FALSE;
	diAPos : DINT;
	diBPos : DINT;
	diCPos : DINT;
	diDPos : DINT;
	diEPos : DINT;
	diFPos : DINT;
	diGPos : DINT;
	diHPos : DINT;
	tyTuning : tyMotionCANTuning;
	diJogVelInUMPS : DINT := 50000;
	diMovePosInUM : DINT := 0;
	diMoveDistInUM : DINT := 0;
	diMoveVelInUMPS : DINT := 50000;
	diMoveAcc : DINT := 500;
	diMoveDec : DINT := 500;
	diMinAbsPosInUM : DINT := -25000;
	diMaxAbsPosInUM : DINT := 10000000;
	bInterruptSensor1 : BOOL;
	bInterruptSensor2 : BOOL;
	bInterruptSensor3 : BOOL;
	bInterruptSensor4 : BOOL;
	bInterruptSensor5 : BOOL;
	bDir : BOOL;
	bNoIndexPulse : BOOL;
	usiNode : USINT;
	sDevice : STRING[3];
	sProgNm : STRING[15] := 'Trav';
	tyParamInHm : tyMotionCANParamInHm;
	tyParamInConvert : tyMotionCANParamInConvert;
	bNtSettingsLoadDone : BOOL := TRUE;
END_VAR
(**)
(*Local*)
VAR
	bRstErr : BOOL;
	udiRstErrOld : UDINT;
	bInitDone : BOOL;
	bInitialDone : BOOL;
	bModuleOKChk : BOOL := FALSE;
	bModuleOK : BOOL;
	bModuleNotOK : BOOL := TRUE;
	bModuleNotOKLock : BOOL;
	bNotInterruptible : BOOL;
	diActualPosInUMOld : DINT;
	usiRstStep : USINT := 0;
	usiStep : USINT;
	usiCount : USINT;
	fbTm : TON := (PT:=T#2s);
	fbServoModuleNotOk : TON := (IN:=FALSE,PT:=T#2s);
	fbServoModuleOk : TON := (IN:=FALSE,PT:=T#5s);
	fbRstNodeTimer : TON := (PT:=T#3s);
	tyParamInMove : tyMotionCANParamInMove;
	tyParamInDriver : tyMotionCANDriverIn := (siModOfOptDisp_6061:=6);
	tyParamOutDriver : tyMotionCANDriverOut;
	fbStop : fbMotionCANStop;
	fbRstAxisErr : fbMotionCANRstAxisErr;
	fbJog : fbMotionCANJog;
	fbMovRel : fbMotionCANMovRel;
	fbMovAbs : fbMotionCANMovAbs;
	fbHoming : fbMotionCANHoming;
	fbPwrOff : fbMotionCANPwrOff;
	fbPwrOn : fbMotionCANPwrOn;
	fbFullHm : fbMotionCANFullHm;
	fbFullMovAbs : fbMotionCANFullMovAbs := (tyInternal:=(fbMotionCANMovAbs:=(tDlyTm:=T#50ms)));
	fbModuleOK : fbMotionCANModuleOK;
	fbSDOWrite : fbCANSDOWriteArrayParam;
	bInletShutterCloseRS : BOOL;
	bOutletShutterCloseRS : BOOL;
	bTravGotoChkPt : BOOL;
	diTravGotoChkPtDist1 : DINT;
	diTravGotoChkPtDist2 : DINT;
	diTravGotoChkPtDist3 : DINT;
	udiModuleNum : UINT := 901;
END_VAR
```

#### Act_Background.st
```iecst
(** 2020-03-16 **)
ACTION Act_Background:

	//Update Parameter
	IF bModuleOK = TRUE THEN

		tyParamInMove.diPosInUM				:= p_diMovePosInUM;
		tyParamInMove.diDistInUM			:= p_diMoveDistInUM;
		tyParamInMove.diVelInUMPS			:= p_diMoveVelInUMPS;
		tyParamInMove.diAcc			:= p_diMoveAcc;
		tyParamInMove.diDec			:= p_diMoveDec;

		fMotionCANUpdtDat(ADR(tyParamOut) , p_tyParamInConvert , tyParamOutDriver , tyParamInDriver , tyParamInMove , p_tyParamInHm , p_bDir, p_eNtParamMotorType);

		bAPosDiff	:= (tyParamOut.bIsHomed = FALSE) OR ((ABS(p_diAPos - tyParamOut.diActualPosInUM)) > 500);
		bBPosDiff	:= (tyParamOut.bIsHomed = FALSE) OR ((ABS(p_diBPos - tyParamOut.diActualPosInUM)) > 500);
		bCPosDiff	:= (tyParamOut.bIsHomed = FALSE) OR ((ABS(p_diCPos - tyParamOut.diActualPosInUM)) > 500);
		bDPosDiff	:= (tyParamOut.bIsHomed = FALSE) OR ((ABS(p_diDPos - tyParamOut.diActualPosInUM)) > 500);
		bEPosDiff	:= (tyParamOut.bIsHomed = FALSE) OR ((ABS(p_diEPos - tyParamOut.diActualPosInUM)) > 500);
		bFPosDiff	:= (tyParamOut.bIsHomed = FALSE) OR ((ABS(p_diFPos - tyParamOut.diActualPosInUM)) > 500);
		bGPosDiff	:= (tyParamOut.bIsHomed = FALSE) OR ((ABS(p_diGPos - tyParamOut.diActualPosInUM)) > 500);
		bHPosDiff	:= (tyParamOut.bIsHomed = FALSE) OR ((ABS(p_diHPos - tyParamOut.diActualPosInUM)) > 500);

		IF p_bDir = TRUE THEN
			bFrontSen	:= tyParamOut.bFwdLmtSen;
			bRearSen	:= tyParamOut.bRevLmtSen;
		ELSE
			bFrontSen	:= tyParamOut.bRevLmtSen;
			bRearSen	:= tyParamOut.bFwdLmtSen;
		END_IF

		CASE p_eNtParamMotorType OF
			DeltaAsdaA2:
				CASE tyParamOut.udiAxisErrID OF
					8976:	sAxisErrTxt	:= 'Over Current';
					12560:	sAxisErrTxt	:= 'Over Voltage';
					12576:	sAxisErrTxt	:= 'Under Voltage';
					12592:	sAxisErrTxt	:= 'Input Power Phase Loss';
					12816:	sAxisErrTxt	:= 'Regeneration Error';
					12848:	sAxisErrTxt	:= 'Overload';
					12849:	sAxisErrTxt	:= 'Pre-overload Warning';
					13056:	sAxisErrTxt	:= 'U,V,W Wiring Error';
					16912:	sAxisErrTxt	:= 'IGBT Temperature Error';
					21296:	sAxisErrTxt	:= 'Memory Error';
					21569:	sAxisErrTxt	:= 'Emergency Stop Activated';
					21570:	sAxisErrTxt	:= 'Forward Limit Switch Error';
					21571:	sAxisErrTxt	:= 'Reverse Limit Switch Error';
					21572:	sAxisErrTxt	:= 'Forward Software Limit';
					21573:	sAxisErrTxt	:= 'Reverse Software Limit';
					21760:	sAxisErrTxt	:= 'DSP Firmware Upgrade';
					25088:	sAxisErrTxt	:= 'CANopen SYNC Error';
					25360:	sAxisErrTxt	:= 'CANopen Data Initial Error';
					25376:	sAxisErrTxt	:= 'Adjustment Error';
					28961:	sAxisErrTxt	:= 'Motor Protection Error';
					28962:	sAxisErrTxt	:= 'Motor Error';
					29445:	sAxisErrTxt	:= 'Encoder Error';
					29446:	sAxisErrTxt	:= 'Encoder Output Error';
					29968:	sAxisErrTxt	:= 'Serial Communication Error';
					29984:	sAxisErrTxt	:= 'Serial Communication Time Out';
					33024:	sAxisErrTxt	:= 'CANbus Error (Bus-off)';
					33040:	sAxisErrTxt	:= 'CANopen SDO receive buffer overrun';
					33056:	sAxisErrTxt	:= 'CANbus Error (Warning)';
					33072:	sAxisErrTxt	:= 'Node Guarding or Heartbeat Error';
					33280:	sAxisErrTxt	:= 'CANopen PDO Object Error';
					33792:	sAxisErrTxt	:= 'Over Speed';
					34304:	sAxisErrTxt	:= 'Abnormal Pulse Control Command';
					34320:	sAxisErrTxt	:= 'Full Closed Loop Excessive Deviation';
					34321:	sAxisErrTxt	:= 'Excessive Deviation';
				END_CASE

			SchneiderLexium28:
				CASE tyParamOut.udiAxisErrID OF
					8724:	sAxisErrTxt	:= 'Over Current';
					8976:	sAxisErrTxt	:= 'Motor Overload';
					8977:	sAxisErrTxt	:= 'Drive overload (foldback)';
					9088:	sAxisErrTxt	:= 'Calculated offsets for current sensors out OF range';
					9089:	sAxisErrTxt := 'Motor phase missing';
					9090:	sAxisErrTxt := 'Overcurrent detected at one OF the digital outputs';
					12560:	sAxisErrTxt	:= 'DC Bus Over Voltage';
					12576:	sAxisErrTxt	:= 'DC Bus Under Voltage';
					12672:	sAxisErrTxt	:= 'Braking Resistor Overload';
					12673:	sAxisErrTxt	:= 'Safety function Safe Torque Off (STO) triggered';
					12674:	sAxisErrTxt	:= 'DC bus voltage measurement';
					12675:	sAxisErrTxt	:= 'Missing mains supply, undervoltage mains supply';
					12676:	sAxisErrTxt := 'The encoder supply voltage has dropped under operational value';
					12677:	sAxisErrTxt := 'The multi turn encoder battery voltage has dropped under 3 Vdc';
					12678:	sAxisErrTxt := 'Internal position synchronization error	detected between the multi turn AND the single turn modules';
					12679:	sAxisErrTxt := 'Generic error code of the multi turn module is detected';
					12697:	sAxisErrTxt := 'Braking resistor overload';
					16512:	sAxisErrTxt	:= 'Drive overtemperature (IPM)';
					16513:	sAxisErrTxt	:= 'Drive overtemperature (controller)';
					16534:	sAxisErrTxt := 'Temperature sensor inoperative';
					17168:	sAxisErrTxt	:= 'Power stage overtemperature';
					17280:	sAxisErrTxt := 'The encoder temperature is too high';
					17424:	sAxisErrTxt	:= 'Motor overtemperature';
					21808:	sAxisErrTxt	:= 'System error detected (nonvolatilememory)';
					21893:	sAxisErrTxt	:= 'Error detected in non-volatile memory';
					21889:	sAxisErrTxt	:= 'System error detected (nonvolatile memory)';
					21890:	sAxisErrTxt	:= 'System error detected (CAN power supply)';
					21891:	sAxisErrTxt	:= 'System error detected (selftest)';
					21894:	sAxisErrTxt	:= 'System error detected (NV ACCESS)';
					25472:	sAxisErrTxt	:= 'Target position rejected';
					25985:	sAxisErrTxt	:= 'System error detected(FPGA)';
					28816:	sAxisErrTxt	:= 'System error detected (FPGA does NOT match firmware)';
					28817:	sAxisErrTxt	:= 'Emergency Stop Activated';
					28961:	sAxisErrTxt := 'Motor blocked';
					29080:	sAxisErrTxt := 'Commutation error detected';
					29568:  sAxisErrTxt	:= 'Error detected in communication with motor encoder';
					29574:	sAxisErrTxt	:= 'Drive is not synchronous wit master cycle';
					29581:	sAxisErrTxt := 'System error detected (encoder)';
					29587:	sAxisErrTxt	:= 'Encoder overvoltage or overcurrent';
					29592:	sAxisErrTxt := 'The returned position value are no longer considered valid';
					29593:	sAxisErrTxt := 'The multi turn encoder requires an explicit configuration command';
					30081:	sAxisErrTxt := 'Target position rejected';
					30082:	sAxisErrTxt := 'No target values received via the fieldbus';
					33072:	sAxisErrTxt	:= 'CANopen: Heartbeat error detected';
					33296:	sAxisErrTxt := 'R_PDO is too short';
					33921:	sAxisErrTxt	:= 'Actual Motor Velocity Too High';
					33553:	sAxisErrTxt	:= 'Motor torque too high FOR an excessive period OF time';
					33664:	sAxisErrTxt := 'Unstable current loop';
					33922:	sAxisErrTxt := 'Velocity deviation too high';
					34321:	sAxisErrTxt	:= 'Position deviation too high';
					34432:	sAxisErrTxt := 'Position deviation via signal output function MC_OK';
					34441:	sAxisErrTxt := 'Position deviation too high (following error)';
					61568:	sAxisErrTxt	:= 'Fieldbus: Communication	error detected';
					65282:	sAxisErrTxt	:= 'Not possible to read data of electronic motor nameplate';
					65296:	sAxisErrTxt	:= 'Forward Limit Switch Error';
					65297:	sAxisErrTxt	:= 'Reverse Limit Switch Error';
					65281:	sAxisErrTxt := 'System error detected';
					65298:	sAxisErrTxt	:= 'Forward Software Limit';
					65299:	sAxisErrTxt	:= 'Reverse Software Limit';
					65301:	sAxisErrTxt := 'The encoder firmware cannot operate on the provided hardware';

				END_CASE

			EstunPronet:
				CASE tyParamOut.udiAxisErrID OF
					65281:	sAxisErrTxt	:= 'Parameter breakdown';//A01
					65282:	sAxisErrTxt	:= 'AD shift channels breakdown';
					65283:	sAxisErrTxt	:= 'Overspeed';
					65284:	sAxisErrTxt	:= 'Overload';
					65285:	sAxisErrTxt := 'Position error counteroverflow ';
					65286:	sAxisErrTxt := 'Position error pulse overflow';
					65287:	sAxisErrTxt	:= 'The setting of electronic gear or given pulse frequency is not reasonable';
					65288:	sAxisErrTxt	:= 'The 1st channel of current detection is wrong.';
					65289:	sAxisErrTxt	:= 'The 2nd channel of current detection is wrong.';
					65290:	sAxisErrTxt	:= 'Incremental Encoder is break off.';//A10
					65292:	sAxisErrTxt	:= 'Overcurrent';
					65293:	sAxisErrTxt	:= 'Overvoltage';
					65294:	sAxisErrTxt	:= 'Undervoltage';
					65295:	sAxisErrTxt := 'Bleeder resistor error';
					65296:	sAxisErrTxt := 'Regeneration error';
					65297:	sAxisErrTxt := 'Resolver error';
					65298:	sAxisErrTxt := 'IGBT superheat alarm';
					65299:	sAxisErrTxt := 'Motor overheat alarm';
					65300:	sAxisErrTxt := 'Power line phase shortage';//A20
					65301:	sAxisErrTxt	:= 'Instantaneous power off alarm';
					65302:	sAxisErrTxt	:= 'Motor temperature detection sensor is break off.';
					65303:	sAxisErrTxt := 'Brake overcurrent alarm';//A23
					65305:	sAxisErrTxt := 'Motor power line U overcurrent';//A25
					65306:	sAxisErrTxt := 'Motor power line V overcurrent';//A26
					65307:	sAxisErrTxt := 'Motor power line W overcurrent';//A27
					65322:	sAxisErrTxt	:= 'Servomotor type error';//A42
					65323:	sAxisErrTxt	:= 'Servo drive type error';
					65325:	sAxisErrTxt	:= 'Absolute encoder multiturn information error';
					65326:	sAxisErrTxt	:= 'Absolute encoder multiturn information overflow';
					65327:	sAxisErrTxt	:= 'Battery voltage below 2.5V';
					65328:	sAxisErrTxt	:= 'Battery voltage below 3.1V';//A48
					65330:	sAxisErrTxt := 'Serial encoder communication overtime ';//A50
					65331:	sAxisErrTxt := 'Absolute encoder overspeed alarm detected';
					65332:  sAxisErrTxt	:= 'Absolute state of serial encoder error';
					65333:	sAxisErrTxt	:= 'Serial encoder calcaution error';
					65334:	sAxisErrTxt := 'Parity bit or end bit in serial encoder control domain error';
					65335:	sAxisErrTxt	:= 'Serial encoder communication data checking error';
					65336:	sAxisErrTxt := 'End bit in serial encoder control domain error';
					65338:	sAxisErrTxt := 'Serial encoder data empty';
					65339:	sAxisErrTxt := 'Serial encoder data format error';
					65340:	sAxisErrTxt := 'Communication module not detected ';//A60
					65341:	sAxisErrTxt := 'Communication unsuccessful';
					65342:	sAxisErrTxt := 'Servo drive can not receive the period data of communication module ';
					65343:	sAxisErrTxt := 'Communication module can not receive the servo drive response data.';
					65344:	sAxisErrTxt := 'Communication module and bus connectionless';
					65346:	sAxisErrTxt := 'CAN communication abnormal';
					65347:	sAxisErrTxt := 'Receiving heartbeat timeout';
					65349:	sAxisErrTxt := 'Synchronization signal monitoring cycle is longer than setting';
					65362: sAxisErrTxt	:= 'Torque output alarm';
				END_CASE
		END_CASE
	ELSE

		tyParamOut.bAxisErr			:= FALSE;
		tyParamOut.bFwdLmtSen		:= FALSE;
		tyParamOut.bInPos			:= FALSE;
		tyParamOut.bIsHomed			:= FALSE;
		tyParamOut.bPosDiff			:= TRUE;
		tyParamOut.bPwrOn			:= FALSE;
		tyParamOut.bRevLmtSen		:= FALSE;
		tyParamOut.bStopped			:= TRUE;
		tyParamOut.diActualPosInUM	:= 0;
		tyParamOut.diHmAcc			:= 0;
		tyParamOut.diHmSpdForSwitch	:= 0;
		tyParamOut.diHmSpdForZero	:= 0;
		tyParamOut.diProfileAcc		:= 0;
		tyParamOut.diProfileDec		:= 0;
		tyParamOut.udiAxisErrID		:= 0;

		bAPosDiff					:= TRUE;
		bBPosDiff					:= TRUE;
		bCPosDiff					:= TRUE;
		bDPosDiff					:= TRUE;
		bEPosDiff					:= TRUE;
		bFPosDiff					:= TRUE;
		bGPosDiff					:= TRUE;
		bHPosDiff					:= TRUE;

	END_IF

	//	Abnormal Movement
	IF eStatus1 <> Error THEN
		IF p_bOps = TRUE AND eStatus = Idle THEN
			IF (ABS(tyParamOut.diActualPosInUM - diActualPosInUMOld) > 2000) AND (ABS(tyParamOut.diActualPosInUM - diActualPosInUMOld) < 30000) THEN
				eStatus1	:= Error;
				udiStatus1	:= 10000;	//Axis Move Abnormally By External Force

				fMotionCANRstCtrlWord(ADR(tyParamOutDriver));
				p_eAct	:= TravActIdle;
				eStat	:= TravActIdle;
			END_IF
		ELSE
			diActualPosInUMOld	:= tyParamOut.diActualPosInUM;
		END_IF
	END_IF

	//Reset Error
	IF (eStatus1 = Error) AND bRstErr THEN
		eStatus1	:= Idle;
		udiStatus1	:= 0;
	END_IF

	//Request Position To Movement Out Of Range
	IF p_bOps
		AND((tyParamInMove.diPosInUM < p_diMinAbsPosInUM) OR (tyParamInMove.diPosInUM > p_diMaxAbsPosInUM))
		AND (eStatus2 <> Error) THEN
		eStatus2	:= Error;
		udiStatus2	:= 10077;	//Request Absolute Position Out Of Range

		fMotionCANRstCtrlWord(ADR(tyParamOutDriver));
		p_eAct	:= TravActIdle;
		eStat	:= TravActIdle;
	END_IF

	//Reset Error
	IF (eStatus2 = Error) AND bRstErr THEN
		eStatus2	:= Idle;
		udiStatus2	:= 0;
	END_IF

	//Sensor Interrupt
	IF bNotInterruptible = TRUE AND eStatus3 <> Error THEN

		IF p_bInterruptSensor1 OR p_bInterruptSensor2 OR p_bInterruptSensor3 OR p_bInterruptSensor4 OR p_bInterruptSensor5 THEN

			eStatus3	:= Error;
			udiStatus3	:= 10041;	//Sensor Interrupt Movement

			fMotionCANRstCtrlWord(ADR(tyParamOutDriver));
			p_eAct	:= TravActIdle;
			eStat	:= TravActIdle;
		END_IF

	END_IF

	//Reset Error
	IF (eStatus3 = Error) AND bRstErr THEN
		eStatus3	:= Idle;
		udiStatus3	:= 0;
	END_IF

	IF bRstErr THEN
		udiStatus	:= 0;
	END_IF

	fbServoModuleOk(IN:= bModuleOK);
	fbServoModuleNotOk(IN:= bModuleOK = FALSE);
	IF fbServoModuleNotOk.Q AND udiStatus <> 10001 THEN

		bModuleNotOK		:= TRUE;
		bModuleNotOKLock	:= TRUE;
		usiRstStep	:= 0;
		tyParamOutDriver.uiCtrlword_6040	:= 0;
		tyParamOutDriver.siModOfOpt_6060	:= 0;
		tyParamOutDriver.diTargetPos_607A	:= 0;
		tyParamOutDriver.udiMoveSpd_6081	:= 0;
		tyParamOutDriver.siHmMethod_6098	:= 0;
		tyParamOutDriver.diJogVel_60FF		:= 0;

		CASE p_eNtParamMotorType OF

			DeltaAsdaA2:
				fbModuleOK(bModuleOK:= FALSE);
				IF eStatus = Idle THEN
					eAct	:= TravActRstNode;
				END_IF

				IF (eStatus = Done OR eStatus = Error)AND eStat = TravActRstNode THEN

					eAct	:= TravActIdle;
				END_IF

			EstunPronet:
				fbModuleOK(bModuleOK:= FALSE);
				IF eStatus = Idle THEN
					eAct	:= TravActRstNode;
				END_IF

				IF (eStatus = Done OR eStatus = Error)AND eStat = TravActRstNode THEN

					eAct	:= TravActIdle;
				END_IF

			SchneiderLexium28:
			// Do Nothing
		END_CASE

	ELSIF bModuleNotOK = TRUE AND fbServoModuleOk.Q THEN

		CASE usiRstStep OF

			0:
				IF eStatus = Idle THEN
					eAct	:= TravActRstAxisErr;
				END_IF

				IF eStatus = Done AND eStat = TravActRstAxisErr THEN
					eAct	:= TravActIdle;
					usiRstStep	:= 4;
				END_IF

			4: tyParamOutDriver.siModOfOpt_6060 := 1;
				usiRstStep	:= 5;

			5: tyParamOutDriver.siModOfOpt_6060 := 1;
				fbRstNodeTimer(IN:=TRUE);

				IF tyParamInDriver.siModOfOptDisp_6061 = 1 THEN
					usiRstStep	:= 6;
					fbRstNodeTimer(IN:=FALSE);
				ELSIF fbRstNodeTimer.Q THEN
					usiRstStep	:= 8;
					fbRstNodeTimer(IN:=FALSE);
				END_IF

			6: tyParamOutDriver.siModOfOpt_6060 := 6;
				fbRstNodeTimer(IN:=FALSE);
				usiRstStep	:= 7;

			7: tyParamOutDriver.siModOfOpt_6060 := 6;
				fbRstNodeTimer(IN:=TRUE);

				IF tyParamInDriver.siModOfOptDisp_6061 = 6 THEN
					usiRstStep	:= 10;
					fbRstNodeTimer(IN:=FALSE);
				ELSIF fbRstNodeTimer.Q THEN
					usiRstStep	:= 9;
					fbRstNodeTimer(IN:=FALSE);
				END_IF

			8:	fbModuleOK(bEn := TRUE, bModuleOK:= FALSE);
				fbRstNodeTimer(IN:=FALSE);
				usiRstStep	:= 9;

			9:	fbModuleOK(bModuleOK:= FALSE);
				IF eStatus = Idle THEN
					eAct	:=TravActRstNode;
				END_IF

				IF eStatus = Done AND eStat = TravActRstNode THEN
					usiRstStep	:= 0;
					eAct		:= TravActIdle;
				END_IF

			10:IF eStatus = Idle THEN
					eAct	:= TravActRstAxisErr;
				END_IF

				IF eStatus = Done AND eStat = TravActRstAxisErr THEN
					eAct			:= TravActIdle;
					usiRstStep	:= 11;
				END_IF

			11:

				IF eStatus = Idle THEN
					eAct	:= TravActSDOWrite;
				END_IF

				IF eStatus = Done AND eStat = TravActSDOWrite THEN
					eAct			:= TravActIdle;
					usiRstStep	:= 13;

				END_IF

			13: bModuleNotOK	:= FALSE;
				usiRstStep	:= 0;
		END_CASE
	ELSE
		eAct	:= TravActIdle;

	END_IF

	IF tyParamOut.bPosDiff = FALSE THEN
		tyParamOutDriver.uiCtrlword_6040.4	:= FALSE;
	END_IF

END_ACTION
```

#### Act_InitGlobal.st
```iecst
(** 2019-04-09 **)
ACTION Act_InitGlobal:

	(* Always Change If Project Change *)

	//Pass Data To Link
	p_bLinkOpsRun ACCESS p_OpsRun;
	p_bLinkStartupRun ACCESS p_StartupRun;
	p_bSimu ACCESS p_UISimuMod;

	p_eLinkMag ACCESS p_NtParamProjMag;
	p_usiLinkMod ACCESS p_ProdRcpCurrRcp1McMod;

	p_diLinkAPos ACCESS p_MagRcpCurrRcpMag1TravPos;
	p_diLinkBPos ACCESS p_MagRcpCurrRcpMag2TravPos;
	p_diLinkCPos ACCESS p_MagRcpCurrRcpMag3TravPos;
	p_diLinkGPos ACCESS p_MagRcpCurrRcpMag4TravPos;

	p_diLinkAPos1 ACCESS p_MagRcpCurrRcpMag1TravPos1;
	p_diLinkBPos1 ACCESS p_MagRcpCurrRcpMag2TravPos1;
	p_diLinkCPos1 ACCESS p_MagRcpCurrRcpMag3TravPos1;
	p_diLinkGPos1 ACCESS p_MagRcpCurrRcpMag4TravPos1;

	p_bLinkNtParamProjRotCylPrep ACCESS p_NtParamProjPullerRotCylPrep;

	p_bLinkOpsTravLifULInDSPos ACCESS p_OpsTravLifULInDSPos;
	p_bLinkOpsTravLifUSMagWidthChk ACCESS p_OpsTravLifLDUSMagWidthChk;

	p_bLinkNtParamProjDsFixToFixRail ACCESS p_NtParamProjDsFixToFixRail;
	p_diLinkFixtoFixPosIn ACCESS p_McParamTravOutletFixtoFixPos;
	p_diLinkMcParamTravPosB ACCESS p_McParamTravPosB;
	p_tyProdRcpCurrRcp ACCESS p_ProdRcpCurrRcp2;

	p_bLinkSafetyRelay ACCESS p_DISafetyRlySig;
	p_bLinkProjLifterMagPlatform ACCESS p_NtParamProjLifterMagPlatform;

		//Trav magwidthCheck
	p_bLinkTravGotoChkPt ACCESS p_OpsTravLifULTravGotoChkPt;
//	p_diLinkTravGotoChkPtDist1 ACCESS p_NtParamTravGotoMagWidthChkPt1;
//	p_diLinkTravGotoChkPtDist2 ACCESS p_NtParamTravGotoMagWidthChkPt2;
//	p_diLinkTravGotoChkPtDist3 ACCESS p_NtParamTravGotoMagWidthChkPt3;
	p_diLinkTravGotoChkPtDist1 ACCESS p_McParamMag1WidthChkDetDist;
	p_diLinkTravGotoChkPtDist2 ACCESS p_McParamMag2WidthChkDetDist;
	p_diLinkTravGotoChkPtDist3 ACCESS p_McParamMag3WidthChkDetDist;

	p_diLaneBOffset ACCESS p_McParamTravLaneBOffset;
	//Pass Data To Internal Use
	p_bEn ACCESS p_DISimServoEn;
	p_udiRstErr ACCESS p_RstErrReset;
	p_bOps ACCESS p_OpsStatusRun;
	p_bManual ACCESS p_UIMnlMod;
//	p_diAPos ACCESS p_MagRcpCurrRcpMag1TravPos;
//	p_diBPos ACCESS p_MagRcpCurrRcpMag2TravPos;
//	p_diCPos ACCESS p_MagRcpCurrRcpMag3TravPos;
	p_diDPos ACCESS p_McParamTravPosA;
//	p_diEPos ACCESS p_McParamTravPosB;
//	p_diGPos ACCESS p_MagRcpCurrRcpMag4TravPos;
	p_tyTuning ACCESS p_NtParamTravTuning;
	p_diJogVelInUMPS ACCESS p_UIMnlTravJogSpd;
	p_diMovePosInUM ACCESS p_UIMnlTravTargetPos;
	p_diMoveDistInUM ACCESS p_UIMnlTravStepSize;
	p_diMoveAcc ACCESS p_NtParamTravAcc;
	p_diMoveDec ACCESS p_NtParamTravDec;
	p_bDir ACCESS p_NtParamTravDir;
	p_usiNode ACCESS p_NtParamTravNode;
	p_sDevice ACCESS p_NtParamTravDevice;
	p_sProgNm ACCESS p_NtParamTravProgNm;
	p_tyParamInHm ACCESS p_NtParamTravParamInHm;
	p_tyParamInConvert ACCESS p_NtParamTravParamInConvert;
	p_bNtSettingsLoadDone ACCESS p_StartupNtSettingsLoadDone;
	p_eNtParamMotorType ACCESS p_NtParamTravMotorType;

	p_bInletShutterCloseRS ACCESS p_DIInShutterCloseRS;
	p_bOutletShutterCloseRS ACCESS p_DIOutShutterCloseRS;
	p_bProjInletShutPrep ACCESS p_NtParamProjInletShutPrep;
//	p_bInShutterDis ACCESS p_McParamInShutterDis;
	p_bProjOutletShutPrep ACCESS p_NtParamProjOutletShutPrep;
	p_bOutShutterDis ACCESS p_McParamOutShutterDis;
	p_bPullerRetSen ACCESS p_DIPullerRetRS;
	p_bPullerExtSen ACCESS p_DIPullerExtRS;
	p_bPullerRotHmRS ACCESS p_DIPullerRotHmRS; //JOHN

	p_bDIConvClrSen ACCESS p_DIConvClrSen;
    p_bDIConvLftSen ACCESS p_DIConvLftSen;
	(* Always Change If Project Change *)

END_ACTION
```

#### Act_Initial.st
```iecst
(** 2020-03-16 **)
ACTION Act_Initial:

	//Initial
	sStatTxt	:= a_sStatText[eStat];

	tyParamInMove.diAcc	:= p_diMoveAcc;
	tyParamInMove.diDec	:= p_diMoveDec;

	fbModuleOK.sDevice	:= p_sDevice;
	fbModuleOK.usiNode	:= p_usiNode;
	fbModuleOK.tDlyTm	:= T#5s;
	fbModuleOK(bEn := FALSE);

	fbSDOWrite.sDevice	:= p_sDevice;
	fbSDOWrite.usiNode	:= p_usiNode;
	fbSDOWrite.eMotorType	:= p_eNtParamMotorType;
	fbSDOWrite(bEn := FALSE);

	fbFullMovAbs.p_tyParamOutDriver		:= ADR(tyParamOutDriver);
	fbFullMovAbs.tyParamInMove.diAcc	:= p_diMoveAcc;
	fbFullMovAbs.tyParamInMove.diDec	:= p_diMoveDec;
	fbFullMovAbs.tyParamInConvert		:= p_tyParamInConvert;
	fbFullMovAbs.bDir					:= p_bDir;
	fbFullMovAbs.bNoIndexPulse			:= p_bNoIndexPulse;
	fbFullMovAbs.eMotorType				:= p_eNtParamMotorType;
	fbFullMovAbs(bEn := FALSE);

	fbFullHm.p_tyParamOutDriver	:= ADR(tyParamOutDriver);
	fbFullHm.bDir				:= p_bDir;
	fbFullHm.bNoIndexPulse		:= p_bNoIndexPulse;
	fbFullHm.eMotorType			:= p_eNtParamMotorType;
	fbFullHm(bEn := FALSE);

	fbPwrOn.p_tyParamOutDriver	:= ADR(tyParamOutDriver);
	fbPwrOn.eMotorType			:= p_eNtParamMotorType;
	fbPwrOn(bEn := FALSE);

	fbPwrOff.p_tyParamOutDriver	:= ADR(tyParamOutDriver);
	fbPwrOff.eMotorType			:= p_eNtParamMotorType;
	fbPwrOff(bEn := FALSE);

	fbHoming.p_tyParamOutDriver	:= ADR(tyParamOutDriver);
	fbHoming.bDir				:= p_bDir;
	fbHoming.bNoIndexPulse		:= p_bNoIndexPulse;
	fbHoming.eMotorType			:= p_eNtParamMotorType;
	fbHoming(bEn := FALSE);

	fbMovAbs.p_tyParamOutDriver		:= ADR(tyParamOutDriver);
	fbMovAbs.tyParamInMove.diAcc	:= p_diMoveAcc;
	fbMovAbs.tyParamInMove.diDec	:= p_diMoveDec;
	fbMovAbs.tyParamInConvert		:= p_tyParamInConvert;
	fbMovAbs.bDir					:= p_bDir;
	fbMovAbs.eMotorType			:= p_eNtParamMotorType;
	fbMovAbs(bEn := FALSE);

	fbMovRel.p_tyParamOutDriver		:= ADR(tyParamOutDriver);
	fbMovRel.tyParamInMove.diAcc	:= p_diMoveAcc;
	fbMovRel.tyParamInMove.diDec	:= p_diMoveDec;
	fbMovRel.tyParamInConvert		:= p_tyParamInConvert;
	fbMovRel.bDir					:= p_bDir;
	fbMovRel.eMotorType			:= p_eNtParamMotorType;
	fbMovRel(bEn := FALSE);

	fbJog.p_tyParamOutDriver	:= ADR(tyParamOutDriver);
	fbJog.tyParamInConvert		:= p_tyParamInConvert;
	fbJog.eMotorType			:= p_eNtParamMotorType;
	fbJog(bEn := FALSE);

	fbRstAxisErr.p_tyParamOutDriver	:= ADR(tyParamOutDriver);
	fbRstAxisErr(bEn := FALSE);

	fbStop.p_tyParamOutDriver	:= ADR(tyParamOutDriver);
	fbStop(bEn := FALSE);

	bModuleNotOK	:= TRUE;
END_ACTION
```

#### Act_InitLocal.st
```iecst
(** 2020-03-16 **)
ACTION Act_InitLocal:

	//Input Reference Link To Local Variable
	p_eAct ACCESS ADR(eAct);
	p_udiRstErr ACCESS ADR(udiRstErr);
	p_bPrep ACCESS ADR(bPrep);
	p_bEn ACCESS ADR(bEn);
	p_bDis ACCESS ADR(bDis);
	p_bOps ACCESS ADR(bOps);
	p_bManual ACCESS ADR(bManual);
	p_diAPos ACCESS ADR(diAPos);
	p_diBPos ACCESS ADR(diBPos);
	p_diCPos ACCESS ADR(diCPos);
	p_diDPos ACCESS ADR(diDPos);
	p_diEPos ACCESS ADR(diEPos);
	p_diFPos ACCESS ADR(diFPos);
	p_diGPos ACCESS ADR(diGPos);
	p_diHPos ACCESS ADR(diHPos);
	p_tyTuning ACCESS ADR(tyTuning);
	p_diJogVelInUMPS ACCESS ADR(diJogVelInUMPS);
	p_diMovePosInUM ACCESS ADR(diMovePosInUM);
	p_diMoveDistInUM ACCESS ADR(diMoveDistInUM);
	p_diMoveVelInUMPS ACCESS ADR(diMoveVelInUMPS);
	p_diMoveAcc ACCESS ADR(diMoveAcc);
	p_diMoveDec ACCESS ADR(diMoveDec);
	p_diMinAbsPosInUM ACCESS ADR(diMinAbsPosInUM);
	p_diMaxAbsPosInUM ACCESS ADR(diMaxAbsPosInUM);
	p_bInterruptSensor1 ACCESS ADR(bInterruptSensor1);
	p_bInterruptSensor2 ACCESS ADR(bInterruptSensor2);
	p_bInterruptSensor3 ACCESS ADR(bInterruptSensor3);
	p_bInterruptSensor4 ACCESS ADR(bInterruptSensor4);
	p_bInterruptSensor5 ACCESS ADR(bInterruptSensor5);
	p_bDir ACCESS ADR(bDir);
	p_bNoIndexPulse ACCESS ADR(bNoIndexPulse);
	p_usiNode ACCESS ADR(usiNode);
	p_sDevice ACCESS ADR(sDevice);
	p_sProgNm ACCESS ADR(sProgNm);
	p_tyParamInHm ACCESS ADR(tyParamInHm);
	p_tyParamInConvert ACCESS ADR(tyParamInConvert);
	p_bNtSettingsLoadDone ACCESS ADR(bNtSettingsLoadDone);

	p_bInletShutterCloseRS ACCESS ADR(bInletShutterCloseRS);
	p_bOutletShutterCloseRS ACCESS ADR(bOutletShutterCloseRS);
	p_bLinkTravGotoChkPt ACCESS ADR(bTravGotoChkPt);
	p_diLinkTravGotoChkPtDist1 ACCESS ADR(diTravGotoChkPtDist1);
	p_diLinkTravGotoChkPtDist2 ACCESS ADR(diTravGotoChkPtDist2);
	p_diLinkTravGotoChkPtDist3 ACCESS ADR(diTravGotoChkPtDist3);

END_ACTION
```

#### Act_Link.st
```iecst
(** 2019-03-29 **)
ACTION Act_Link:

	IF p_eLinkMag = LDMagQuadruple THEN
		CASE p_usiLinkMod OF
			0: //LDModLoadLnA:
				p_diAPos := p_diLinkAPos;
				p_diBPos := p_diLinkBPos;
				p_diCPos := p_diLinkCPos;
				p_diGPos := p_diLinkGPos;

			1: //LDModLoadLnB:
				p_diAPos := p_diLinkAPos1;
				p_diBPos := p_diLinkBPos1;
				p_diCPos := p_diLinkCPos1;
				p_diGPos := p_diLinkGPos1;

			2: //LDModLoadLnAB:
				p_diAPos := p_diLinkAPos;
				p_diBPos := p_diLinkBPos;
				p_diCPos := p_diLinkCPos1;
				p_diGPos := p_diLinkGPos1;
		END_CASE
	ELSE
		IF p_bLinkTravGotoChkPt THEN // To Check the Magazine Width - Offset of Traverser
			p_diAPos := p_diLinkAPos + p_diLinkTravGotoChkPtDist1;
			p_diBPos := p_diLinkBPos + p_diLinkTravGotoChkPtDist2;
			p_diCPos := p_diLinkCPos + p_diLinkTravGotoChkPtDist3;
		ELSE
			p_diAPos := p_diLinkAPos;
			p_diBPos := p_diLinkBPos;
			p_diCPos := p_diLinkCPos;
			p_diGPos := p_diLinkGPos;
		END_IF
	END_IF

	IF p_bManual = TRUE THEN
		p_diMoveVelInUMPS ACCESS p_UIMnlTravNomSpd;
	ELSE
		p_diMoveVelInUMPS ACCESS p_NtParamTravAutoSpd;
	END_IF

	IF p_bLinkNtParamProjRotCylPrep	= FALSE THEN
		IF (p_bProjInletShutPrep = TRUE) AND p_bLinkOpsTravLifULInDSPos = FALSE THEN
			IF p_bInletShutterCloseRS = FALSE OR p_bPullerRetSen = FALSE OR p_bPullerExtSen
				THEN
				p_bInterruptSensor1 := TRUE;
			ELSE
				p_bInterruptSensor1 := FALSE;
			END_IF
		ELSE
			p_bInterruptSensor1 := FALSE;
		END_IF

		IF p_bProjOutletShutPrep = TRUE AND p_bOutShutterDis = FALSE AND p_bLinkOpsTravLifULInDSPos = FALSE THEN
			IF p_bOutletShutterCloseRS = FALSE OR p_bPullerRetSen = FALSE OR p_bPullerExtSen
				THEN
				p_bInterruptSensor2 := TRUE;
			ELSE
				p_bInterruptSensor2 := FALSE;
			END_IF
		ELSE
			p_bInterruptSensor2 := FALSE;
		END_IF
	ELSE
		IF (p_bProjInletShutPrep = TRUE) AND p_bLinkOpsTravLifULInDSPos = FALSE AND p_bLinkOpsTravLifUSMagWidthChk = FALSE THEN
			IF p_bInletShutterCloseRS = FALSE OR p_bPullerRetSen = FALSE OR p_bPullerExtSen
				THEN
					p_bInterruptSensor1 := TRUE;
			ELSE
					p_bInterruptSensor1 := FALSE;
			END_IF
		ELSE
			p_bInterruptSensor1 := FALSE;
		END_IF

		IF p_bProjOutletShutPrep = TRUE AND p_bOutShutterDis = FALSE AND p_bLinkOpsTravLifULInDSPos = FALSE
			AND p_bLinkProjLifterMagPlatform = FALSE // rotate w/ platform
			THEN
			IF p_bOutletShutterCloseRS = FALSE OR p_bPullerRetSen = FALSE OR p_bPullerExtSen
				THEN
				p_bInterruptSensor2 := TRUE;
			ELSE
				p_bInterruptSensor2 := FALSE;
			END_IF
		ELSE
			p_bInterruptSensor2 := FALSE;
		END_IF
	END_IF

	p_bInterruptSensor3 := p_bDIConvClrSen OR p_bDIConvLftSen;//p_bLinkSafetyRelay = FALSE;

	p_bInterruptSensor4 := p_bPullerRetSen = FALSE OR p_bPullerExtSen OR p_bPullerRotHmRS = FALSE;

	IF p_bLinkNtParamProjDsFixToFixRail THEN
		p_diEPos := p_diDPos + p_diLinkFixtoFixPosIn - p_tyProdRcpCurrRcp.diWidthInUM + p_diLaneBOffset;
	ELSE
		p_diEPos := p_diLinkMcParamTravPosB;
	END_IF

END_ACTION
```

#### Act_LinkAction.st
```iecst
(** 2019-10-21 **)
ACTION Act_LinkAction:

	IF eStatus = Idle THEN
		IF bModuleNotOK THEN
			p_eAct ACCESS ADR(eAct);
		ELSE
			IF p_bLinkStartupRun = TRUE THEN
				p_eAct ACCESS p_StartupTravAct;
			ELSIF p_bLinkOpsRun = TRUE THEN
				p_eAct ACCESS p_OpsTravLifLDTravAct;
			ELSIF p_bManual = TRUE OR p_bSimu THEN
				p_eAct ACCESS p_UITravAct;
			ELSE
				p_eAct ACCESS ADR(eAct);
			END_IF
		END_IF
	END_IF

	IF EDGENEG(p_bManual) OR EDGENEG(p_bLinkOpsRun) OR EDGENEG(p_bLinkStartupRun) THEN
		tyParamOutDriver.uiCtrlword_6040	:= 0;
	END_IF

END_ACTION
```

#### Init.st
```iecst
(** 2019-04-24 **)
PROGRAM _INIT

	(* Always Change If Project Change *)

	//Pass Address To Global Address For External Use
	//Action, State & Status
	p_TravStat		:= ADR(eStat);
	p_TravStatus	:= ADR(eMainStatus);
	p_TravStatTxt	:= ADR(sStatTxt);

	//Alarm
	p_TravAlmData	:= ADR(tyAlmData);
	p_TravAlmData1	:= ADR(tyAlmData1);
	p_TravAlmData2	:= ADR(tyAlmData2);
	p_TravAlmData3	:= ADR(tyAlmData3);

	//Output
	p_TravParamOut		:= ADR(tyParamOut);
	p_TravPwrOn			:= ADR(tyParamOut.bPwrOn);
	p_TravIsHomed		:= ADR(tyParamOut.bIsHomed);
	p_TravPosDiff		:= ADR(tyParamOut.bPosDiff);
	p_TravAxisErr		:= ADR(tyParamOut.bAxisErr);
	p_TravAxisErrID		:= ADR(tyParamOut.udiAxisErrID);
	p_TravFwdLmtSen		:= ADR(tyParamOut.bFwdLmtSen);
	p_TravRevLmtSen		:= ADR(tyParamOut.bRevLmtSen);
	p_TravActualPos		:= ADR(tyParamOut.diActualPosInUM);
	p_TravAxisErrTxt	:= ADR(sAxisErrTxt);
	p_TravAPosDiff		:= ADR(bAPosDiff);
	p_TravBPosDiff		:= ADR(bBPosDiff);
	p_TravCPosDiff		:= ADR(bCPosDiff);
	p_TravDPosDiff		:= ADR(bDPosDiff);
	p_TravEPosDiff		:= ADR(bEPosDiff);
	p_TravFPosDiff		:= ADR(bFPosDiff);
	p_TravGPosDiff		:= ADR(bGPosDiff);
	p_TravHPosDiff		:= ADR(bHPosDiff);
	p_TravJogging		:= ADR(bJogging);
	p_TravFrontSen		:= ADR(bFrontSen);
	p_TravRearSen		:= ADR(bRearSen);

	(* Always Change If Project Change *)

END_PROGRAM
```

### Program Logical/CANOpenServo/Lifter/LifterBtm (IEC) - 1.00.0 - NtMotion v5.00.0

#### InputRef.var
```iecst
(*2020-03-16*)
(**)
(*General*)
VAR
	p_eAct : REFERENCE TO eLifterAction;
	p_udiRstErr : REFERENCE TO UDINT;
	p_bPrep : REFERENCE TO BOOL;
	p_bEn : REFERENCE TO BOOL;
	p_bDis : REFERENCE TO BOOL;
END_VAR
(**)
(*Configuration*)
VAR
	p_bOps : REFERENCE TO BOOL;
	p_bManual : REFERENCE TO BOOL;
	p_diGoASlt : REFERENCE TO DINT;
	p_diASltToSltDist : REFERENCE TO DINT;
	p_diASlt1Pos : REFERENCE TO DINT;
	p_diGoBSlt : REFERENCE TO DINT;
	p_diBSltToSltDist : REFERENCE TO DINT;
	p_diBSlt1Pos : REFERENCE TO DINT;
	p_diGoCSlt : REFERENCE TO DINT;
	p_diCSltToSltDist : REFERENCE TO DINT;
	p_diCSlt1Pos : REFERENCE TO DINT;
	p_diGoDSlt : REFERENCE TO DINT;
	p_diDSltToSltDist : REFERENCE TO DINT;
	p_diDSlt1Pos : REFERENCE TO DINT;
	p_diAPos : REFERENCE TO DINT;
	p_diBPos : REFERENCE TO DINT;
	p_diCPos : REFERENCE TO DINT;
	p_diDPos : REFERENCE TO DINT;
	p_diEPos : REFERENCE TO DINT;
	p_diFPos : REFERENCE TO DINT;
	p_diGPos : REFERENCE TO DINT;
	p_diHPos : REFERENCE TO DINT;
	p_tyTuning : REFERENCE TO tyMotionCANTuning;
	p_diJogVelInUMPS : REFERENCE TO DINT;
	p_diMovePosInUM : REFERENCE TO DINT;
	p_diMoveDistInUM : REFERENCE TO DINT;
	p_diMoveVelInUMPS : REFERENCE TO DINT;
	p_diMoveAcc : REFERENCE TO DINT;
	p_diMoveDec : REFERENCE TO DINT;
	p_diMinAbsPosInUM : REFERENCE TO DINT;
	p_diMaxAbsPosInUM : REFERENCE TO DINT;
	p_bInterruptSensor1 : REFERENCE TO BOOL;
	p_bInterruptSensor2 : REFERENCE TO BOOL;
	p_bInterruptSensor3 : REFERENCE TO BOOL;
	p_bInterruptSensor4 : REFERENCE TO BOOL;
	p_bInterruptSensor5 : REFERENCE TO BOOL;
	p_bInterruptSensor6 : REFERENCE TO BOOL;
	p_bDir : REFERENCE TO BOOL;
	p_bNoIndexPulse : REFERENCE TO BOOL;
	p_usiNode : REFERENCE TO USINT;
	p_sDevice : REFERENCE TO STRING[3];
	p_sProgNm : REFERENCE TO STRING[15];
	p_tyParamInHm : REFERENCE TO tyMotionCANParamInHm;
	p_tyParamInConvert : REFERENCE TO tyMotionCANParamInConvert;
	p_bNtSettingsLoadDone : REFERENCE TO BOOL;
	p_eNtParamMotorType : REFERENCE TO eServoMotorType;
	p_bUITeachServo : REFERENCE TO BOOL;
	p_bPullerRetSen : REFERENCE TO BOOL;
	p_bPullerExtSen : REFERENCE TO BOOL;
	p_bOutletShutterCloseRS : REFERENCE TO BOOL;
	p_bProjInletShutPrep : REFERENCE TO BOOL;
	p_bProjOutletShutPrep : REFERENCE TO BOOL;
	p_bInletShutterCloseRS : REFERENCE TO BOOL;
	p_bOutShutterDis : REFERENCE TO BOOL;
	p_bDIConvClrSen : REFERENCE TO BOOL;
	p_bDIConvLftSen : REFERENCE TO BOOL;
END_VAR
```

#### InputRef_Link.var
```iecst
(*2019-04-09*)
(**)
(*External*)
VAR
	p_bLinkOpsRun : REFERENCE TO BOOL;
	p_bLinkStartupRun : REFERENCE TO BOOL;
END_VAR
(**)
VAR
	p_diLinkSltToSltDist : REFERENCE TO DINT;
	p_bLinkDILifterTimingBeltSen : REFERENCE TO BOOL;
	p_bLinkDILifterSafetyLmtSW1 : REFERENCE TO BOOL;
	p_bLinkDILifterSafetyLmtSW2 : REFERENCE TO BOOL;
	p_diLinkSltToSltDist1 : REFERENCE TO DINT;
END_VAR
(**)
VAR
	p_eLinkMag : REFERENCE TO eLDMag;
	p_usiLinkMod : REFERENCE TO USINT;
END_VAR
(**)
VAR
	p_diLinkASlt1Pos : REFERENCE TO DINT;
	p_diLinkBSlt1Pos : REFERENCE TO DINT;
	p_diLinkCSlt1Pos : REFERENCE TO DINT;
	p_diLinkDSlt1Pos : REFERENCE TO DINT;
	p_diLinkASlt1Pos1 : REFERENCE TO DINT;
	p_diLinkBSlt1Pos1 : REFERENCE TO DINT;
	p_diLinkCSlt1Pos1 : REFERENCE TO DINT;
	p_diLinkDSlt1Pos1 : REFERENCE TO DINT;
	p_bLinkNtParamProjRotCylPrep : REFERENCE TO BOOL;
	p_bLinkOpsTravLifULInDSPos : REFERENCE TO BOOL;
	p_bLinkSafetyRelay : REFERENCE TO BOOL;
	p_bLinkProjLifterMagPlatform : REFERENCE TO BOOL;
END_VAR
```
